		(*Wrap up break Flags to Variable for shipment to UI*)
		ECatSlave_Cable_Breaks.0:= ATV320_NotPresent AND Prev_EcatNode_Present;
		ECatSlave_Cable_Breaks.1:= ATV320_PortB_MissingLink;


(*$$$$$$$$$$$$$$$$$$$$$$$$$$$$$$$$$$$$$$$$$$$$$$$$$$$$Gather All Standard and System Inputs $$$$$$$$$$$$$$$$$$$$$$$$$$$$$$$$$$$$$$$$$$$$$$$$$$$$$$$$$$$$$*)

	(*--------------- System Inputsfrom VFD System Outputs -------------------------*)

	(*Status_Word*)
		Operating_State_Ready:= NOT Status_Word.0;
		Operating_State_Switched_On:=Status_Word.1;
		Operating_State_Operation_enabled:=Status_Word.2;
		Operating_State_Fault:=Status_Word.3;
		Voltage_Enabled:=Status_Word.4;
		Operating_State_Quick_Stop:=Status_Word.5;
		Operating_State_Switch_On_Dissabled:=Status_Word.6;
		Error_Class0:=Status_Word.7;
		Halt_Requested:=Status_Word.8;
		Remote:=Status_Word.9;
		Target_Reached:=Status_Word.10;
		Internal_Limit:=Status_Word.11;
		Operating_Mode_Specific:=Status_Word.12;
		X_ERR:=Status_Word.13;
		X_End:=Status_Word.14;
		Ref_OK:=Status_Word.15;



(*$$$$$$$$$$$$$$$$$$$$$$$$$$$$$$$$$$$$$$$$$$$$$$$$$$ Internal Code $$$$$$$$$$$$$$$$$$$$$$$$$$$$$$$$$$$$$$$$$$$$$$$$$$$$$$$$*)


	(*Capture time between part feeding*)
	Move_TMR(
			IN:= (Enable_Operation AND NOT Operating_State_Switch_On_Dissabled) AND Enable_Motion,
			PT:= T#9999s,
			Q=> ,
			ET=>
			);
	IF Move_TMR.IN
		THEN
			Move_TIME:= Move_TMR.ET;
	END_IF;


(*$$$$$$$$$$$$$$$$$$$$$$$$$$$$$$$$$$$$$$$$$$$$$$ Transfer Standard Outputs $$$$$$$$$$$$$$$$$$$$$$$$$$$$$$$$$$$$$$$$$$$*)

	Discrete_Image.Status_Word:= Status_Word;
	Discrete_Image.Control_Word:= Control_Word;
	Discrete_Image.Target_Velocity:= Target_Velocity;
	Discrete_Image.ECAT_Cable_Breaks:= ECatSlave_Cable_Breaks;

	Discrete_Image.VFD_State:= VFD_State;
	Discrete_Image.Move_TIME:= Move_TIME;



	(*--------------- System Outputs to VFD System Inputs -------------------------*)

	(*Control Word*)
	Control_Word.0:= (Operating_State_Switch_On AND NOT Operating_State_Switch_On_Dissabled) AND Enable_Motion;
	Control_Word.1:= Enable_Voltage AND Enable_Motion;
	Control_Word.2:= Operating_State_Quick_Stop_Req;
	Control_Word.3:= (Enable_Operation AND NOT Operating_State_Switch_On_Dissabled) AND Enable_Motion;
	Control_Word.4:= Operating_Mode_Bit4;
	Control_Word.5:= Operating_Mode_Bit5;
	Control_Word.6:= Operating_Mode_Bit6;
	Control_Word.7:= Fault_Reset;
	Control_Word.8:= Halt;
	Control_Word.9:= Operating_Mode_Bit9;
	Control_Word.10:= FALSE; (*reserved - must be 0*)
	Control_Word.11:= FALSE; (*reserved - must be 0*)
	Control_Word.12:= FALSE; (*reserved - must be 0*)
	Control_Word.13:= FALSE; (*reserved - must be 0*)
	Control_Word.14:= FALSE; (*reserved - must be 0*)
	Control_Word.15:= FALSE; (*reserved - must be 0*)


	(*Output Frequency*)
	IF (Requested_Freq>=0) AND (Requested_Freq<51)
		THEN
			Target_Velocity:= (Requested_Freq * 30);
	ELSE
			Target_Velocity:= 0;
	END_IF;
















(*end*)

END_FUNCTION_BLOCK

// ---- POUs/FBs/FB_GTAC_Ped_20240808.TcPOU
(*!!!!!!!!!!!!!!!!!!!!!!!!!!!!!!!!!!!!!!!!!!!!!!!!!!!!!!!!!!!!!!!!!!!!!!!!!!!!!!!!!!!!!!!!!!!!!!!!!!!!!!!!!!!!!!!!!!!!!!!!!!!!!!!!!!!!!!!!!!!!!!!!!!!!!!!!!!
FB for framework of a generic Ped Station (welding, Sealing, stud welding etc)
	author: Brent Lekx-Toniolo of Sodecia GTAC
	Feb, 2015
--------------------------------------------------------------------------------------------------------------
REVISION NOTES:
	Version: 20150224:
	- Original Concept, b.lekx-toniolo
	Version: 20150426:
	- Change Order of Fix ID, b.lekx-toniolo
	- Added Complete Reset Input
	Version: 20151104:
	- added linkable hardware types, b.lekx-toniolo
	Version: 20160728
	- added control fro brake option, b.lekx-toniolo
	- added configuration inputs for Input node and VB counts, b.lekx-toniolo
	Version: 20160915
	- added "blank_position_checks" Input, b.lekx-toniolo, r.remillard, j.vandongen
	- added "Dresser_Enable" Input, b.lekx-toniolo, r.remillard, j.vandongen
	Version: 20160926
	- Corrected doubled up valve 1 instance, b.lekx-toniolo
	Version 20170404
	- add Part present sensors, j.vandongen
	Version 20170704
	- changed valve instances, j.vandongen
	Version 20170725
	- added VB_Node_Count to UI and updated discrete_image, j.vandongen
	- removed dresser wording form variables to make fb more generic, j.vandongen
	- moved tool_at_positions to outside the fb, j.vandongen
	Version 20170810
	- corrected PP fault issue, j.vandongen
	Version 20220808
	- Added Prev_EcatNode_Present and Prev_EcatNode_ID, c.drees
	Version 20230126
	- Built in SwingArm functionality to combine PEDxx with SwingArmXX, c.drees
	Version 20240514
	- Add in Nodelayout configuration data area, b.lexk-toniolo
	Version 20240808
	- Add in ability to externally control portions of the N50 output block
--------------------------------------------------------------------------------------------------------------
*)

FUNCTION_BLOCK FB_GTAC_Ped_20240808
	VAR_INPUT

		Enable_Prog: BOOL;
		Enable_Motion: BOOL;
		Mode_Select: INT;
		Go_Home: BOOL;
		Reset_Production: BOOL;
		Model_Data: INT;
		Task_Data: UINT;
		Manual_Requests: DINT;
		Dry_Cycle: BOOL;
		Cell_In_Services: BOOL;
		PrevProcess_Complete: BOOL;
		Blank_Position_Checks: BOOL;
		Start_TipDress_Cycle: BOOL;
		Start_TipChange_Cycle: BOOL;
		
		(*Generic Position Variables*)
		Tool_At_Home: BOOL;
		Tool_At_Work0: BOOL;
		Tool_At_Work1: BOOL;

		Part_Present1_REQ: BOOL;
		Part_Present2_REQ: BOOL;
		Part_Present3_REQ: BOOL;
		Part_Present4_REQ: BOOL;

		Work_Robots_Clear: BOOL;
		Work_Robots_WorkingOK: BOOL;
		Work_Robots_Complete: BOOL;
		Work_Robots_LHPartInEOAT: BOOL;
		Work_Robots_RHPartInEOAT: BOOL;
		Work_Robots_CommonPartInEOAT: BOOL;
		Work_Robots_EOATEmpty: BOOL;
	(*Node Counts and configuration data*)
		Input_Node_Count: UDINT;
		Output_Node_Count: UDINT;
			Output_Node_UserREQS: UINT;
		VB_Node_Count: UDINT;
		Part_Present_Count: UDINT;
		Option_SwingCylinder: BOOL;		(*Enables a Cylinder used for changing the Ped Item (Weld gun as example) position OR Tip Dress Swing*)
			Swing_ADV_REQ: BOOL;		
			Swing_RET_REQ: BOOL;
		Option_TipDresser: BOOL;	(*Enables Tip Dresser functionality*)
		Option_TipChanger: BOOL;		(*Enables Tip Changer functionality*)
		NodeLayout:udt_ECATNodeData_20221507;

	(*Ecat configuration*)
	
		Prev_EcatNode_Present:BOOL;
		Prev_EcatNode_ID:STRING;
	END_VAR

	VAR
(*Hardware Related Data Types*)
			(*Develop "Beckhoff Nodes"*)
			{attribute 'OPC.UA.DA':='1'}
			N01 AT %I*: udt_EP1008_002_v2;
			{attribute 'OPC.UA.DA':='1'}
			N02 AT %I*: udt_EP1008_002_v2;
			{attribute 'OPC.UA.DA':='1'}
			N50 AT %Q*: udt_EP2028_002_v2;
			{attribute 'OPC.UA.DA':='1'}
			N50_STAT AT %I*: udt_EP2028_002_STAT;
			{attribute 'OPC.UA.DA':='1'}
			N100 AT %Q*: udt_SMC_EX260_ValveBank;
			{attribute 'OPC.UA.DA':='1'}
			N100_STAT AT %I*:udt_SMC_EX260_Stat;
(* Nodes States*)
		NodeState: ARRAY[0..63] OF UINT;
		DiscreteNode_OK: BOOL;
(*Cable Break States*)
		ECatSlave_Cable_Breaks: ARRAY[0..1] OF DINT;
(*Standard Internal Variables*)

		(*Generic Position Variables*)
		Tool_At_Work: UINT;

		(*General Internals*)
		In_Auto: BOOL;
		In_Manual: BOOL;

		Auto_Run: BOOL;
		Reset_All_Completes:BOOL;

		Start_Work_Robots: BOOL;
		Work_Robots_Proceed: BOOL;

		Prod_Inc: R_TRIG;
		Cycle_Time: TON;
		Cycle_Time_Pulse: R_TRIG;
		CLFaulted: UDINT;
		PPFaulted: UDINT;
		Manual_Ind_HomePrompt: BOOL;

(*Non-Standard Variables*)
		(*FB Instances*)
		Swing1FB: FB_Cylinder_Status;
		Part_Present1FB: FB_PP_Sensor;
		Part_Present2FB: FB_PP_Sensor;
		Part_Present3FB: FB_PP_Sensor;
		Part_Present4FB: FB_PP_Sensor;

		(*Valve FBs*)
		Valve1FB: FB_GTAC_Valve_20170704;
		Valve2FB: FB_GTAC_Valve_20170704;
		(*Tool Positions*)
		Swing1ADVD: BOOL;
		Swing1RETD: BOOL;
		(*Motion Sequence Variables*)
			Clamp_Step: UINT;
			Repo1_Step: UINT;
			Repo2_Step: UINT;
			Repo3_Step: UINT;
			Repo4_Step: UINT;
			Unclamp_Step: UINT;


END_VAR

	(*data that needs to be retained in the event of a power cycle*)
	VAR PERSISTENT
		Working_Complete: BOOL;
		Cycle_Complete: BOOL;
		Production_Count:INT;
		TipDress_Complete: BOOL;
		TipChange_Complete: BOOL;
		Repo_REQS: UINT;
	END_VAR

	VAR_OUTPUT
		Prog_Ok: BOOL;
		Discrete_Image: udt_PEDxx_Image_20240808;
		In_Auto_Mode: BOOL;
		In_Manual_Mode: BOOL;
		Manual_Indicators: DINT;
		At_Home: BOOL;
		CLFaults1:UDINT;
		CLFaults2:UDINT;
		CLFaults3:UDINT;
		CLFaults4:UDINT;
		PPFaults: UDINT;
		Prod_Count_Out: INT;
		Cycle_Time_Out: TIME;
		PrevCycle_Time_Out: TIME;
		Tool_Call_ForWorkRobots: BOOL;
		Robots_Clear_ToProceed: BOOL;
		Task_ID: UINT;
		Fix_ID: UINT;
		Model_ID: UINT;
		Work_Complete_Ack: BOOL;
		Repo_Ack: UINT;

	(*Part Present Sensors*)
		(*Main Body Present*)
		Part_Present1: BOOL;
		Part_Present2: BOOL;
		Part_Present3: BOOL;
		Part_Present4: BOOL;

	END_VAR

	(*Set FB_OK to True*)
	Prog_OK:= TRUE;
(*$$$$$$$$$$$$$$$$$$$$$$$$$$$$$$$$$$$$$$$$$$$$$$$$Gather Status Of Hardware $$$$$$$$$$$$$$$$$$$$$$$$$$$$$$$$$$$$$$$$$$$$$$$$$$$$*)
	(*Discrete I/O Nodes*)
	IF N01.InfoData.State=8 OR (Input_Node_Count<1)
		AND (N02.InfoData.State=8 OR (Input_Node_Count<2))
		AND (N50_STAT.InfoData.State=8 OR (Output_Node_Count<1))
		AND (N100_Stat.InfoData.State=8 OR (VB_Node_Count<1))
			THEN DiscreteNode_OK:=TRUE;
	ELSE DiscreteNode_OK:=FALSE;
	END_IF;
	
	(*Cable Break Detection*)
	ECatSlave_Cable_Breaks[0]:= FUN_GTAC_EcatSlaveConnState
							(N01.InfoData.State,
							N02.InfoData.State,
							N50_STAT.InfoData.State,
							N100_Stat.InfoData.State,
							0,0,0,0,0,0,0,0,0,0,0,0,0,0,0,0,0,0,0,0,0,0,0,0,0,0); (*Function Returns Flags to warn of possible cable break*)

(*$$$$$$$$$$$$$$$$$$$$$$$$$$$$$$$$$$$$$$$$$$$$$ Gather Safety Inputs $$$$$$$$$$$$$$$$$$$$$$$$$$$$$$$$$$$$$$$$$$$$$$$$$$$$$$$$$*)

(*$$$$$$$$$$$$$$$$$$$$$$$$$$$$$$$$$$$$$$$$$$$$$ Gather Standard Inputs $$$$$$$$$$$$$$$$$$$$$$$$$$$$$$$$$$$$$$$$$$$$$$$$$$$$$$$$$*)
	IF Option_SwingCylinder
		THEN
		(*Swing1 - Ped item OR Tip Dresser Swing (if Option_TipDresser is enabled)*)
		Swing1FB(
			Advanced_Sensor:= N01.I.0,
			Retracted_Sensor:= N01.I.1,
			Advance_Solenoid:= N100.Q.0,
			Retract_Solenoid:= N100.Q.1,
			Adv_Delay:= T#0.5S ,
			Ret_Delay:= T#0.5s ,
			Fault_Delay:= T#4s ,
			In_Advanced_Position=> Swing1ADVD,
			In_Retracted_Position=> Swing1RETD,
			Faulted=> CLFaults1.0 );
	ELSIF NOT  Option_SwingCylinder
		THEN
		Swing1ADVD:= FALSE;
		Swing1RETD:= TRUE;
		CLFaults1.0:= FALSE;

	END_IF;

(*$$$$$$$$$$$$$$$$$$$$$$$$$$$$$$$$$$$$$$$$$$$$$$$$ Internal Code $$$$$$$$$$$$$$$$$$$$$$$$$$$$$$$$$$$$$$$$$$$$$$$$$$$$$$$$$$$$$$$$$$$$*)
(*Auto / Manual Mode Code*)
In_Auto:= TRUE;(*FORCED IN AUTO*)

	IF Mode_Select.0 AND NOT Mode_Select.1
		THEN
			In_Auto:= TRUE;
			In_Auto_Mode:= TRUE;
	END_IF;
	IF NOT Mode_Select.0 AND Mode_Select.1
		THEN
			In_Auto:= FALSE;
			In_Auto_Mode:= FALSE;
	END_IF;
	In_Manual:= NOT In_Auto;
	In_Manual_Mode:= In_Manual;

(*--------------------------------------------------------------------------------Tool Positions---------------------------------------------------------------*)
(*+++++++++++THIS AREA IS CUSTOM PER INSTALLATION AND WILL HAVE TO BE MODIFIED PER +++++++++++++*)
(*+++++++++++THIS AREA IS CUSTOM PER INSTALLATION AND WILL HAVE TO BE MODIFIED PER +++++++++++++*)

	Tool_At_Work.0:= Tool_At_Work0;
	Tool_At_Work.1:= Tool_At_Work1;

(*>>>>>>>>>>>>>>>>>>>>>>>>>>>>>>>>>>>>>>>>>> Auto Run Cycle >>>>>>>>>>>>>>>>>>>>>>>>>>>>>>>>>>>>>>>*)
(*+++++++++++THIS AREA IS CUSTOM PER INSTALLATION AND WILL HAVE TO BE MODIFIED PER +++++++++++++*)
(*+++++++++++THIS AREA IS CUSTOM PER INSTALLATION AND WILL HAVE TO BE MODIFIED PER +++++++++++++*)
	(*Control of Auto_Run*)
	Auto_Run:= Enable_Motion AND In_Auto AND Model_Data<>0 AND NOT Cycle_Complete;

	(*Auto Run Enables All Other Auto Cycle Code*)
	IF Auto_Run
		THEN
			IF NOT Working_Complete  AND PrevProcess_Complete
				THEN
					(*Start Work Robots*)
					Start_Work_Robots:= (Work_Robots_CommonPartInEOAT OR Work_Robots_LHPartInEOAT OR Work_Robots_RHPartInEOAT)
										AND (((Tool_At_Work.0 AND NOT Repo_Reqs.0) OR (Tool_At_Work.1 AND Repo_Reqs.0)) OR Blank_Position_Checks)
										AND (Model_Data <> 0);
;					(*Allow Work Robots To Proceed*)
					Work_Robots_Proceed:= (Work_Robots_CommonPartInEOAT OR Work_Robots_LHPartInEOAT OR Work_Robots_RHPartInEOAT)
										AND Tool_At_Work.0 AND NOT Repo_Reqs.0 AND PrevProcess_Complete;
			ELSE
					Start_Work_Robots:= FALSE;
					Work_Robots_Proceed:= FALSE;
			END_IF;

	ELSE
		Start_Work_Robots:= FALSE;
	END_IF;

(*---------------------------------------------------------------Completes----------------------------------------------------*)
	(*Wrok at Ped Complete*)
	IF Work_Robots_Complete
		THEN
		Working_Complete:= TRUE;
	END_IF;

(*!!!!!!!!!!!!!!!!!!!!!!!!!!!!!!!!!!!!!!!!!!!!!!!!!!!!!!!!!!!!!!!!!!!!!!!!!!!!!!!!!!!!!!!!!!!!!!!!! Cycle Complete !!!!!!!!!!!!!!!!!!!!!!!!!!!!!!!!!!!!!!!!!!!!!!!!!!!!!!!!!!!!!!!!!!!!!!!!!!!!!!!!!!!!!!!!!!*)
	(*Set Cycle Complete*)
	IF Auto_Run AND Working_Complete
		THEN Cycle_Complete:= TRUE;
	END_IF;
	(*Reset All Completes*)
	IF Work_Robots_Clear
		THEN
			IF Work_Robots_EOATEmpty
				THEN
					Reset_All_Completes:= TRUE;
			ELSE
					Reset_All_Completes:= FALSE;
			END_IF;
	END_IF;
	(*Perform Actual Reset*)
		IF Reset_All_Completes
			THEN
				Cycle_Complete:= FALSE;
				Working_Complete:= FALSE;
				Reset_All_Completes:= FALSE;
		END_IF;


(*$$$$$$$$$$$$$$$$$$$$$$$$$$$$$$$$$$$ Production Counter $$$$$$$$$$$$$$$$$$$$$$$$$$$$$$$$$$$$$$$$$$*)
	(*Increment Production Counter*)
	Prod_Inc.CLK:= Cycle_Complete;
	Prod_Inc();
	IF Prod_Inc.Q
		THEN
		Production_Count:= Production_Count+1;
	END_IF;
	IF Reset_Production
		THEN
		Production_Count:= 0;
	END_IF;
	Prod_Count_Out:= Production_Count;
(*~~~~~~~~~~~~~~~~~~~~~~~~~~~~~~~~ Cycle Time Counters ~~~~~~~~~~~~~~~~~~~~~~~~~*)
	(*Move Previous To Register*)
	Cycle_Time_Pulse.CLK:= Cycle_Complete;
	Cycle_Time_Pulse();
	IF Cycle_Time_Pulse.Q
		THEN
		PrevCycle_Time_Out:= Cycle_Time_Out;
	END_IF;
	(*Monitor Current Cycle Time*)
		Cycle_Time.PT:= T#9999S;
		Cycle_Time.IN:= NOT Cycle_Time_Pulse.Q ;
		Cycle_Time();
		Cycle_Time_Out:= Cycle_Time.ET;


(*%%%%%%%%%%%%%% Call Robots to Tool and Give Them, Task ID, Fixture ID and Model ID %%%%%%%%%%%%%%%%%*)

	(* Perform Call To Tool*)
	Tool_Call_ForWorkRobots:= Enable_Motion AND (NOT Cell_In_Services OR NOT Work_Robots_Clear)
	 							AND Start_Work_Robots;

	(*Allow Robots to Proceed Into Tool*)
	(*!!!!!This is the final OK to allow Robots Into the Tool Area, So it Better Be Ready!!!!!!!*)
	IF Enable_Motion
		THEN
			IF Work_Robots_Proceed AND Work_Robots_WorkingOK
				THEN Robots_Clear_ToProceed:=TRUE;
			END_IF;
		ELSE Robots_Clear_ToProceed:= FALSE;
	END_IF;

	(*Develop Task IDs - See Global Variable, "TaskID_Record"*)

	IF Start_Work_Robots AND Enable_Motion
		THEN Task_ID:= Task_Data;
	ELSE Task_ID:= 0;
	END_IF;

	(*Develop Fixture ID*)
	IF Work_Robots_CommonPartInEOAT AND NOT Work_Robots_LHPartInEOAT AND NOT Work_Robots_RHPartInEOAT
		THEN
			Fix_ID:= 1;
	ELSIF Work_Robots_LHPartInEOAT AND NOT Work_Robots_RHPartInEOAT AND NOT Work_Robots_CommonPartInEOAT
		THEN
			Fix_ID:= 2;
	ELSIF NOT Work_Robots_LHPartInEOAT AND Work_Robots_RHPartInEOAT AND NOT Work_Robots_CommonPartInEOAT
		THEN
			Fix_ID:= 3;
	ELSE
			Fix_ID:= 0;
	END_IF;
	(*Develop Model ID*)
	Model_ID:=Model_Data;

(*+++++++++++++++++++++++++++++++++++++++++++++++ Task Complete Acks ++++++++++++++++++++++++++*)

	(*Weld Complete Ack*)
	Work_Complete_Ack:= Work_Robots_Complete AND Working_Complete;



(*!!!!!!!!!!!!!!!!!!!!!!!!!!!!!!!!!!!!!!!!!!!!!!!!!!!!!!!!!!!!!!!!!!!!!!!!!!!!!!!!!!!!!!!! Tool Repositions !!!!!!!!!!!!!!!!!!!!!!!!!!!!!!!!!!!!!!!!!!!!!!!!!!!!!!!!!!!!!!!!!!!!!!!!!!!!!!!!!!!!!!!!!!!*)
(*+++++++++++THIS AREA IS CUSTOM PER INSTALLATION AND WILL HAVE TO BE MODIFIED PER +++++++++++++*)
(*+++++++++++THIS AREA IS CUSTOM PER INSTALLATION AND WILL HAVE TO BE MODIFIED PER +++++++++++++*)

	(*Reposition Request#1*)
	IF FALSE
		THEN
			Repo_Reqs.0:= TRUE;
	END_IF;
	(*Reposition Request#2*)
	IF FALSE
		THEN
			Repo_Reqs.1:= TRUE;
	END_IF;
	(*Reposition Request#3*)
	IF FALSE
		THEN
			Repo_Reqs.2:= TRUE;
	END_IF;
	(*Reposition Request#4*)
	IF FALSE
		THEN
			Repo_Reqs.3:= TRUE;
	END_IF;
	(*Reset All Reposition Acks At the End Of Cycle*)
	IF Cycle_Complete
		THEN
			Repo_Reqs:= 0;
	END_IF;
(*------------------------- Reposition Acks ---------------------*)
	Repo_Ack.0:= Repo_Reqs.0 AND FALSE;
	Repo_Ack.1:= Repo_Reqs.0 AND FALSE;
	Repo_Ack.2:= Repo_Reqs.0 AND FALSE;
	Repo_Ack.3:= Repo_Reqs.0 AND FALSE;



(*?????????????????????????????????????????????????????????????????????????????????????????????????????????????????????????????????*)

(*$$$$$$$$$$$$$$$$$$$$$$$$$$$$$$$$$$$$$$$$$$$$$$$$$$$ Faults $$$$$$$$$$$$$$$$$$$$$$$$$$$$$$$$$$$$$$$$$$$$$$$$$$$$$$$*)
	(*Clamp/Cylider Faults Group 1*)
		IF CLFaults1>0
			THEN CLFaulted.1:=TRUE;
		ELSE
			CLFaulted.1:=FALSE;
		END_IF;
	(*Clamp/Cylider Faults Group 2*)
		IF CLFaults2>0
			THEN CLFaulted.2:=TRUE;
		ELSE
			CLFaulted.2:=FALSE;
		END_IF;
	(*Clamp/Cylider Faults Group 3*)
		IF CLFaults3>0
			THEN CLFaulted.3:=TRUE;
		ELSE
			CLFaulted.3:=FALSE;
		END_IF;
	(*Clamp/Cylinder Faults Group 4 - Reserved Flag for QA Check Motion Faults*)
		IF CLFaults4>0
			THEN CLFaulted.4:=TRUE;
		ELSE
			CLFaulted.4:=FALSE;
		END_IF;
	(*Bit 0 is designated as ANY Clamp Group Faulted*)
	IF CLFaulted.1 OR CLFaulted.2 OR CLFaulted.3
		THEN CLFaulted.0:= TRUE;
	ELSE CLFaulted.0 := FALSE;
	END_IF;

	(*Part Present Sensor Faults*)
		IF PPFaults>0
			THEN PPFaulted.0:=TRUE;
		ELSE
			PPFaulted.0:=FALSE;
		END_IF;

(*$$$$$$$$$$$$$$$$$$$$$$$$$$$$$$$$$$$$$$$$$$$$$$ Transfer Standard Outputs $$$$$$$$$$$$$$$$$$$$$$$$$$$$$$$$$$$$$$$$$$$*)

	(*Transfer General Status and I/O Images for Display On UI*)
	Discrete_Image.Input_Node_Count:= Input_Node_Count;
	Discrete_Image.Output_Node_Count:= Output_Node_Count;
	Discrete_Image.VB_Node_Count:= VB_Node_Count;
	Discrete_Image.Option_SwingCylinder:= Option_SwingCylinder;
	Discrete_Image.Option_TipDresser:= Option_TipDresser;
	Discrete_Image.Option_TipChanger:= Option_TipChanger;
	
	Discrete_Image.CLFaults1:= CLFaults1;
	Discrete_Image.CLFaults2:= CLFaults2;
	Discrete_Image.CLFaults3:= CLFaults3;
	Discrete_Image.CLFaults4:= CLFaults4;
	Discrete_Image.CLFaulted:= CLFaulted;
	
	Discrete_Image.PPFaults:= PPFaults;
	Discrete_Image.PPFaulted:= PPFaulted;
	
	
	Discrete_Image.N01:= N01;
	Discrete_Image.N02:= N02;
	Discrete_Image.N50_STAT:= N50_STAT;
	Discrete_Image.N50:= N50;
	Discrete_Image.N100_STAT:= N100_STAT;
	Discrete_Image.N100:= N100;

	Discrete_Image.NodeLayout:= NodeLayout;
	
	
(*-----------------------------------------------------------------------------------------Transfer Discrete Outputs --------------------------------------------------------------------------------*)

	(*N50 Output Block*)
	IF Enable_Motion AND (Output_Node_Count >0) THEN
		IF Option_TipDresser THEN
			N50.Q.0:= FALSE;		(*Dedicated for Dresser Cutter CW*)
			N50.Q.1:= FALSE;		(*Dedicated for Dresser Cutter CCW*)
			N50.Q.2:= Output_Node_UserREQS.2;
			N50.Q.3:= Output_Node_UserREQS.3;
			N50.Q.4:= Output_Node_UserREQS.4;
			N50.Q.5:= Output_Node_UserREQS.5;
			N50.Q.6:= Output_Node_UserREQS.6;
			N50.Q.7:= Output_Node_UserREQS.7;
		ELSE
			N50.Q.0:= Output_Node_UserREQS.0;
			N50.Q.1:= Output_Node_UserREQS.1;
			N50.Q.2:= Output_Node_UserREQS.2;
			N50.Q.3:= Output_Node_UserREQS.3;
			N50.Q.4:= Output_Node_UserREQS.4;
			N50.Q.5:= Output_Node_UserREQS.5;
			N50.Q.6:= Output_Node_UserREQS.6;
			N50.Q.7:= Output_Node_UserREQS.7;
		END_IF;
	ELSE
		N50.Q:= 0;	
	END_IF;
	
	
(*-----------------------------------------------------------------------------------------Transfer Valve Outputs --------------------------------------------------------------------------------*)

	(*Valve 1, A+B*)
	(*Swing Cylinder 1*)
		Valve1FB
			(
			Enable_Motion:= Enable_Motion AND Option_SwingCylinder,
			Enable_Latch:= TRUE,					(*Enabling Runs Valve as detent type (maintained solenoids*)
			Enable_SideA_PreCharge:= FALSE,		(*Enabling Turns Side A PreCharge Active, reset when Side B is energized in Auto*)
			Enable_SideB_PreCharge:= FALSE,		(*Enabling Turns Side B PreCharge Active, reset when Side A is energized in Auto*)
			PreCharge_Time:= T#0.1S,
			Enable_Auto_Commands:= In_Auto,
			In_Auto_SideA_Command:= Swing_ADV_REQ,
			In_Auto_SideB_Command:= Swing_RET_REQ ,
			Enable_Manual_Commands:= In_Manual,
			In_Manual_SideA_Command:= FALSE,
			In_Manual_SideB_Command:= FALSE,
			SideA_Indicator:= Tool_At_Work.0,
			SideB_Indicator:= Tool_At_Work.1,
			TurnOn_SideA_SOL=> N100.Q.0,
			TurnOn_SideB_SOL=> N100.Q.1,
			TurnOn_SideA_Indicator=> Manual_Indicators.0,
			TurnOn_SideB_Indicator=> Manual_Indicators.1
			 );


(*$$$$$$$$$$$$$$$$$$$$$$$$$$$$$$$$$$$$$$$$$$$$$$ Transfer Safety Outputs $$$$$$$$$$$$$$$$$$$$$$$$$$$$$$$$$$$$$$$$$$$*)

END_FUNCTION_BLOCK

// ---- POUs/FBs/FB_Cylinder_Status.TcPOU
(*FB for replacement of typical clamp fault checking code":
	Original Author(s): Brent Lekx-Toniolo of Toniolo Research & Development Inc.; 
	August 2010; version 3.0


------------------------------------------------------------------------------------------
REVISION NOTES:
	Version 20170615
		-  Added disable fault input, b.lekx-toniolo / j.bysma

------------------------------------------------------------------------------------------
*)
FUNCTION_BLOCK FB_Cylinder_Status

	VAR_INPUT
		Enable_FB: BOOL;
		Advanced_Sensor: BOOL;
		Retracted_Sensor: BOOL;
		Advance_Solenoid: BOOL;
		Retract_Solenoid: BOOL;
		Adv_Delay: TIME;
		Ret_Delay: TIME;
		Fault_Delay: TIME;
		Disable_Fault: BOOL;
	END_VAR

	VAR
		At_Advanced: BOOL;
		At_Retracted: BOOL;
		Adv_Delay_TMR: TON;
		Ret_Delay_TMR: TON;
		Sensor_FLT_TMR: TON;
		Advancing_FLT_TMR: TON;
		Retracting_FLT_TMR: TON;
	END_VAR

	VAR_OUTPUT
		FB_OK: BOOL;
		In_Advanced_Position: BOOL;
		In_Retracted_Position: BOOL;
		Faulted: BOOL;
		Sensor_Fault: BOOL;
		Advancing_Fault: BOOL;
		Retracting_Fault: BOOL;
	END_VAR

	(*Set FB_OK to True*)
	FB_OK:= TRUE;
(*$$$$$$$$$$$$$$$$$$$$$$$$$$$$$$$$$$ Internal Code $$$$$$$$$$$$$$$$$$$$$$$$$$$$$$$$$$$$$$$$$$$$$$$*)
	(*Develop Advanced Position*)
	At_Advanced:=Advanced_Sensor AND NOT Retracted_Sensor;

	(*Develop Retracted Position*)
	At_Retracted:=Retracted_Sensor AND NOT Advanced_Sensor;

	(*Delay Advanced Position Output*)
	Adv_Delay_TMR.PT:=Adv_Delay;
	Adv_Delay_TMR.IN:=At_Advanced;
	Adv_Delay_TMR();
	In_Advanced_Position:=Adv_Delay_TMR.Q;

	(*Delay Retracted Position Output*)
	Ret_Delay_TMR.PT:=Ret_Delay;
	Ret_Delay_TMR.IN:=At_Retracted;
	Ret_Delay_TMR();
	In_Retracted_Position:=Ret_Delay_TMR.Q;

(*$$$$$$$$$$$$$$$$$$$$$$$$$$$$$$$$$$$$$$$$ Fault Code $$$$$$$$$$$$$$$$$$$$$$$$$$$$$$$$$$$$$$$$$$$$$$$$*)
	(*Sensor Fault*)
	Sensor_FLT_TMR.PT:=Fault_Delay;
	Sensor_FLT_TMR.IN:=(NOT At_Advanced AND NOT At_Retracted) OR (At_Advanced AND At_Retracted);
	Sensor_FLT_TMR();
	Sensor_Fault:=Sensor_FLT_TMR.Q;

	(*Advancing Fault*)
	Advancing_FLT_TMR.PT:=Fault_Delay;
	Advancing_FLT_TMR.IN:=Advance_Solenoid AND NOT At_Advanced AND NOT Sensor_Fault;
	Advancing_FLT_TMR();
	Advancing_Fault:=Advancing_FLT_TMR.Q;

	(*Retracting Fault*)
	Retracting_FLT_TMR.PT:=Fault_Delay;
	Retracting_FLT_TMR.IN:=Retract_Solenoid AND NOT At_Retracted AND NOT Sensor_Fault;
	Retracting_FLT_TMR();
	Retracting_Fault:=Retracting_FLT_TMR.Q;

	(*Develop Fault Output*)
	Faulted:= NOT Disable_Fault AND (Sensor_Fault OR Advancing_Fault OR Retracting_Fault);

END_FUNCTION_BLOCK

// ---- POUs/FBs/FB_PP_Sensor.TcPOU
(*FB for replacement of typical part present sesnors fault checking
	Original Author(s):. Brent Lekx-Toniolo of Toniolo Research & Development Inc.; 
	August 2010; version 2.0*)


FUNCTION_BLOCK FB_PP_Sensor
VAR_INPUT
		Enable_FB: BOOL;
		Sensor_Input: BOOL;
		On_Trigger1: BOOL;
		On_Trigger2: BOOL;
		Off_Trigger1: BOOL;
		Off_Trigger2: BOOL;
		Disable_Faults: BOOL;
		Fault_Delay: TIME;
END_VAR
VAR
		NotON_FLT_TMR: TON;
		NotOFF_FLT_TMR: TON;

END_VAR

VAR_OUTPUT
		FB_OK: BOOL;
		Status: BOOL;
		Faulted: BOOL;
		NotON_Fault: BOOL;
		NotOFF_Fault: BOOL;
END_VAR

	(*Set FB_OK to True*)
	FB_OK:= TRUE;
(*$$$$$$$$$$$$$$$$$$$$$$$$$$$$$$$$$$ Internal Code $$$$$$$$$$$$$$$$$$$$$$$$$$$$$$$$$$$$$$$$$$$$$$$*)
	(*Pass Status Straight Thru*)
	Status:= Sensor_Input;

	(*Pass Faults*)
	Faulted:= NotON_Fault OR NotOff_Fault;

	(*Develop Not On When Required Fault*)
	NotOn_FLT_TMR.PT:= Fault_Delay;
	NotOn_FLT_TMR.IN:= On_Trigger1 AND On_Trigger2 AND NOT Sensor_Input AND NOT Disable_Faults;
	NotOn_FLT_TMR();
	NotOn_Fault:= NotOn_FLT_TMR.Q;

	(*Develop Not Off When Required Fault*)
	NotOff_FLT_TMR.PT:= Fault_Delay;
	NotOff_FLT_TMR.IN:= Off_Trigger1 AND Off_Trigger2 AND Sensor_Input AND NOT Disable_Faults;
	NotOff_FLT_TMR();
	NotOff_Fault:= NotOff_FLT_TMR.Q;

END_FUNCTION_BLOCK

// ---- POUs/FBs/FB_GTAC_Valve_20170704.TcPOU
(*FB for use with standard double sided Solenoid Valve:
	Original Author(s): Brent Lekx-Toniolo of Sodecia GTAC; 
------------------------------------------------------------------------------------------
REVISION NOTES:
	Version 20150218
	- Original Concept, b.lekx-toniolo (S.H.H.D.I.)
	Version 20160407
	- Added Enable Latch (Detent Type) functionality, r.remillard
	Version 20170704
	-incorporated precharge into the function block, j.vandongen

------------------------------------------------------------------------------------------
*)


FUNCTION_BLOCK FB_GTAC_Valve_20170704

VAR_INPUT
	Enable_Motion: BOOL;
	Enable_Auto_Commands: BOOL;
	Enable_Latch: BOOL;									(*Used to maintain Solenoid at last requested state*)
	Enable_SideA_PreCharge: BOOL;
	Enable_SideB_PreCharge: BOOL;
	In_Auto_SideA_Command: BOOL;
	In_Auto_SideB_Command: BOOL;
	Enable_Manual_Commands: BOOL;
	In_Manual_SideA_Command: BOOL;
	In_Manual_SideB_Command: BOOL;
	SideA_Indicator: BOOL;
	SideB_Indicator: BOOL;
	PreCharge_Time: TIME;
END_VAR

VAR
	In_Auto_SideA_REQ: BOOL;
	In_Auto_SideB_REQ: BOOL;
	In_Manual_SideA_REQ: BOOL;
	In_Manual_SideB_REQ: BOOL;
	PreCharge_Timer_SideA: TON;
	PreCharge_Timer_SideB: TON;
END_VAR

VAR_OUTPUT
	TurnOn_SideA_SOL: BOOL;
	TurnOn_SideB_SOL: BOOL;
	TurnOn_SideA_Indicator: BOOL;
	TurnOn_SideB_Indicator: BOOL;

END_VAR

(*Gather Auto Mode Requests*)
	In_Auto_SideA_REQ:= Enable_Motion AND Enable_Auto_Commands AND In_Auto_SideA_Command;
	In_Auto_SideB_REQ:= Enable_Motion AND Enable_Auto_Commands AND In_Auto_SideB_Command;



(*Gather Manual Mode Requests*)
	In_Manual_SideA_REQ:= Enable_Motion AND Enable_Manual_Commands AND In_Manual_SideA_Command;
	In_Manual_SideB_REQ:= Enable_Motion AND Enable_Manual_Commands AND In_Manual_SideB_Command;



(*Pre Charge Timers*)
	PreCharge_Timer_SideA(
					In:= Enable_SideA_PreCharge AND (In_Auto_SideA_REQ OR (PreCharge_Timer_SideA.Q AND NOT In_Auto_SideB_REQ)),
					PT:= PreCharge_Time
					);

	PreCharge_Timer_SideB(
					In:= Enable_SideB_PreCharge AND (In_Auto_SideB_REQ OR (PreCharge_Timer_SideA.Q AND NOT In_Auto_SideA_REQ)),
					PT:= PreCharge_Time
					);



(*Set Actual Outputs*)
	(*Valve Outputs*)
	TurnOn_SideA_SOL:= (((In_Auto_SideA_REQ AND (PreCharge_Timer_SideA.Q OR NOT Enable_SideA_PreCharge))
						OR (In_Auto_SideB_REQ AND NOT PreCharge_Timer_SideB.Q AND Enable_SideB_PreCharge)
						OR In_Manual_SideA_REQ)
						OR (Enable_Latch AND TurnOn_SideA_SOL AND NOT (In_Auto_SideB_REQ OR In_Manual_SideB_REQ)))
						AND NOT TurnOn_SideB_SOL;

	TurnOn_SideB_SOL:= (((In_Auto_SideB_REQ AND (PreCharge_Timer_SideB.Q OR NOT Enable_SideB_PreCharge))
						OR (In_Auto_SideA_REQ AND NOT PreCharge_Timer_SideA.Q AND Enable_SideA_PreCharge)
						 OR In_Manual_SideB_REQ)
						OR (Enable_Latch AND TurnOn_SideB_SOL AND NOT (In_Auto_SideA_REQ OR In_Manual_SideA_REQ)))
						AND NOT TurnOn_SideA_SOL;



	(*Indicator Outputs*)
	TurnOn_SideA_Indicator:= SideA_Indicator;
	TurnOn_SideB_Indicator:= SideB_Indicator;



















(*end*)

END_FUNCTION_BLOCK

// ---- POUs/FBs/FB_VertiGuard_20260310.TcPOU

FUNCTION_BLOCK FB_VertiGuard_20260310

VAR_INPUT
	
		Enable_FB: BOOL;
		Enable_Motion: BOOL;
		Enable_Latch: BOOL;

		GateClose_REQ: BOOL;		(*Request to close the door*)
		GateOpen_REQ: BOOL;			(*Request to open the door*)
		
		GateOpened_Time: TIME;		(*Door Open Fault Control Timer*)
		GateClosed_Time: TIME;		(*Door Closed Fault Control Timer*)
		
		GateOpen_Precharge_Time: TIME;	(*Pre Charge Time For Opening Gate*)

		GateClosed_Switches: BOOL;	(*Switches to detect Door Closed*)
		GateOpened_Switches: BOOL;	(*Switches to detect Door opened*)

		Fault_Time: TIME;
		
END_VAR

VAR
	
		Gate_CloseSR: SR; 					(*Latch to Close the door*)
		Gate_OpenSR: SR;					(*Latch to Open the door*)

		GateOpen_Precharge_TMR: TON; 		(*Pre Charge Timer For Opening The Gate*)
		GateOpened_TMR: TON;				(*Timer to say gate is open, no door open switches*)
		GateClosed_TMR: TON;				(*Timer to say gate is closed*)

		Fault_TMR: TON;

END_VAR

VAR_OUTPUT

		FB_OK: BOOL;

		GateClose_CMD: BOOL;	(*Command the door to close*)
		GateOpen_CMD: BOOL;		(*Command the door to open*)
		Gate_Closed: BOOL;		(*Door is closed*)
		Gate_Opened: BOOL;		(*Door is open*)

		Faulted: BOOL;	

END_VAR

(*Set FB_OK to True*)
	FB_OK:= TRUE;

	(*Set Gate to Close*)
	Gate_CloseSR(
			SET1:= Enable_Latch AND GateClose_REQ AND NOT GateOpen_REQ,
			RESET:= NOT Enable_Latch OR (GateOpen_REQ AND Gate_Closed),
			Q1=>
			);

	(*Set Gate to Open*)
	Gate_OpenSR(
			SET1:= Enable_Motion AND Enable_Latch AND GateOpen_REQ AND NOT GateClose_REQ,
			RESET:= NOT Enable_Motion OR NOT Enable_Latch OR (GateClose_REQ OR Gate_Opened),
			Q1=>
			);

	(*Pre Charge Timer For Opening Guard*)
	GateOpen_Precharge_TMR(
					In:= Enable_Motion AND ((Enable_Latch AND Gate_OpenSR.Q1) OR (NOT Enable_Latch AND GateOpen_REQ)),
					PT:= GateOpen_Precharge_Time
					);

	(*Set Actual Outputs*)
	(*Valve Outputs*)
	(*Note ------> The closed state has a pin lock so at the moment the gate is closed, we cancel the latch*)
	GateClose_CMD:= (((Enable_Latch AND Gate_CloseSR.Q1 (*AND NOT Gate_Closed*)) OR (NOT Enable_Latch AND GateClose_REQ)) AND NOT ((Enable_Latch AND Gate_OpenSR.Q1) OR (NOT Enable_Latch AND GateOpen_REQ)))
					OR (((Enable_Latch AND Gate_OpenSR.Q1) OR (NOT Enable_Latch AND GateOpen_REQ)) AND NOT GateOpen_Precharge_TMR.Q);
	GateOpen_CMD:= Enable_Motion AND GateOpen_Precharge_TMR.Q AND ((Enable_Latch AND Gate_OpenSR.Q1) OR (NOT Enable_Latch AND GateOpen_REQ)) AND NOT ((Enable_Latch AND Gate_CloseSR.Q1) OR (NOT Enable_Latch AND GateClose_REQ));
					
	(*Gate Opened Timer*)
	GateOpened_TMR(
			IN:= GateOpened_Switches AND GateOpen_CMD,
			PT:= GateOpened_Time,
			Q=> ,
			ET=>
			);

	(*Gate Closed Timer*)
	GateClosed_TMR(
			IN:= GateClosed_Switches,
			PT:= GateClosed_Time,
			Q=> ,
			ET=>
			);

	(*Capture Gate Status*)
	IF GateClosed_Switches AND GateClosed_TMR.Q
		THEN
			Gate_Closed:= TRUE;
			Gate_Opened:= FALSE;
	ELSIF GateOpened_Switches AND GateOpened_TMR.Q
		THEN
			Gate_Closed:= FALSE;
			Gate_Opened:= TRUE;
	END_IF;
	
	(*Capture Gate Faults*)
	Fault_TMR(
			IN:= (GateClose_CMD AND NOT Gate_Closed) OR (GateOpen_CMD AND NOT Gate_Opened),
			PT:= Fault_Time,
			Q=> Faulted,
			ET=> );


(*end*)

END_FUNCTION_BLOCK

// ---- POUs/GTAC_CONFIG.TcPOU
(* FOR USE BY SODECIA GTAC ONLY !!!*)
(* Sodecia GTAC Configuration data for this particular machine*)

(*----------------------------------------------------------------------------------------------------------------------
REVISION NOTES: 
	Date: Dec 2019
	- Added PROD_CONFIG action and modified production code for R&D request, b.lekx-toniolo/r.remillard
	Date: Jan 2021
	- Automated Machine Serial Variable, b.lekx-toniolo
	Date: Oct 2021
	- Updated serial section for new engineering serial format changes, b.lekx-toniolo
	Date: Feb 2024
	- Added In_Sim_Mode for simulation integration, b.lekx-toniolo
	Date: Sept 2024
	- Added MD component, b.lekx-toniolo
	Date: November 2024
	- PD to IS rename, as per GH SSCC610 repo Issue#162, b.lekx-toniolo

------------------------------------------------------------------------------------------------------------------------*)



PROGRAM GTAC_CONFIG
VAR
		(*Machine Specific Information: Serial Number, Comon Name, Build Level Used, Application Devloper*)
		Machine_Serial: STRING;
		Machine_Common_Name: STRING;
		Machine_Build_Used: STRING;
		Machine_Appl_Dev: STRING;
		
		(*Production Reporting Configuration Data*)
		ProdConfig_Target_CycleTime: TIME;
		ProdConfig_Common: udt_Generic_ShiftCommonConfig_20220420;
		ProdConfig_Day: udt_Generic_ShiftConfigTOD_20160527;
		ProdConfig_Aft: udt_Generic_ShiftConfigTOD_20160527;
		ProdConfig_Mid: udt_Generic_ShiftConfigTOD_20160527;

		ProdConfig_OK: BOOL;
		ProdConfig_Source_FLT: BOOL;
		ProdConfig_Option_SelectInShiftChange: BOOL;

		(*Config Data (For Use to Configure Code Directives)*)
		Option_EL6900_TemperatureHighLimit: INT;

		Option_Air1: BOOL;
		Option_Air2: BOOL;

		Option_Water1: BOOL;
		Option_Water2: BOOL;

		Option_WaterTimeOut_Enable: BOOL;
		Option_WaterFlowTimeOut_SP: TIME;
		Option_WaterTempHighLimit1: REAL;
		Option_WaterFlowLowLimit1: REAL;
		Option_WaterTempHighLimit2: REAL;
		Option_WaterFlowLowLimit2: REAL;

		Option_ESW_Count: UINT;

		Option_IS_Count: UINT;
		Option_IC_Count: UINT;
		Option_HumanFix_Enables: UDINT;
		Option_InternalFix_Count: UINT;
		Option_Robot_Count: UINT;
		Option_Ped_Count: UINT;
		Option_StudController_Count: UINT;
		Option_SealController_Count: UINT;
		Option_NutWelder_Count: UINT;
		(*Option_EOAT_Count: UINT;*)
		Option_LaserController_Count: UINT;
		Option_SD_Count: UINT;
		Option_MD_Count: UINT;
		Option_VFD_Count: UINT;
		Option_EP9214_Count: UINT;
		(*General Development State Modes for Cell*)
		Dry_Cycle_Enabled: BOOL;			(*Place Machine Into Dry Cycle (Ignore PP Sensors)*)
		Local_DryCycle_Enables: UDINT;	(*Used to place individual fixtures into Dry Cycle*)
		Low_Speed_Enabled: BOOL;		(*Set All Robots and Drives to Low Speed Mode*)
		Under_Construction: BOOL; 			(*Set Machine Into Construction Mode for Easier Teaching Etc !!!! Use with Caution !!!!*)
		In_SIM_Mode: BOOL;					(*Set machine into Sim mode during simulation development*)


		(*Configuration Fault Flag*)
		Fault: UDINT;


	Report_Trigger_ACKS: INT;
END_VAR

(*$$$$$$$$$$$$ Set Data As required to configure the machine $$$$$$$$$$$$$$$$$$$$*)

(*-----------------------------------------Machine / Application Specific Information-----------------------------------*)

(*NOTE: Machine Serial is now automatically read from the project name, simply rename your project elements for your machine and we'll do the rest!*)
	Machine_Serial:= FUN_GTAC_ReturnSetLengthSTR(Out_To_ICxx.Appdata.ProjectName, 22);

(*NOTE: Change to a common use name that the customer will recognize*)
	Machine_Common_Name:= 'Volvo Truck V2004 Front Bumper';
	
(*NOTE: When you started with a server copy of the FW the software came in a folder called All_yyymmdd_state*) 
	(*use this for below and change the value below only once upon creating this application, this takes a snap shot of the FW build level you started with*)
	Machine_Build_Used:= 'All_20250506_release';
	
(*NOTE: Be sure to Enter your name or initials here, if mulitple application developers worked on the project then list all*)
	Machine_Appl_Dev:= 'w.griffiths, r.jone, b.lekx-toniolo';
		

(*---------------------------------------Production Report Configuration -----------------------------------*)
(*Machine Target Cycle Time (can also be set individually at each fixture, see Fixture -> Production Action*)
(*Changes per Model ID - All controlled by Fixture 01*)

(*504*)
	IF (Fix01.Model_ID=1) THEN
		ProdConfig_Target_CycleTime:=T#156S;
(*524*)
	ELSIF (Fix01.Model_ID=2) THEN
		ProdConfig_Target_CycleTime:=T#184.8S;
(*543*)
	ELSIF (Fix01.Model_ID=3) THEN
		ProdConfig_Target_CycleTime:=T#136.1S;
(*526 OR 536*)
	ELSIF (Fix01.Model_ID=4) OR (Fix01.Model_ID=5) THEN
		ProdConfig_Target_CycleTime:=T#221S;
(*550 OR 571*)
	ELSIF (Fix01.Model_ID=6) OR (Fix01.Model_ID=7) THEN
		ProdConfig_Target_CycleTime:= T#251S;
	END_IF
	
	

(*Call Prod_Config_Constraints Action*)
	PROD_CONFIG_Constraints();

(*Call Prod_Config Action*)
	PROD_CONFIG();
	
(*Call Reports Action*)
	REPORTS();	

(*Call SIM Action*)
	SIM();	

(*-----------------------------------------Machine Configuration Options -----------------------------------*)
(*Select to Check for 1st MAIN Air Manifold Faults*)
	Option_Air1:= TRUE;
(*Select to Check for 2nd MAIN Air Manifold Faults*)
	Option_Air2:= FALSE;

(*Select to Check for 1st MAIN Water Manifold Faults*)
	Option_Water1:= FALSE;
(*Select to Check for 2nd MAIN Water Manifold Faults*)
	Option_Water2:= FALSE;

(*Global Water Setpoints*)
	Option_WaterTimeOut_Enable:= NOT Under_Construction AND
									TRUE;		(*Enable Robot Water Flow Timeout Feature (Stop Water flow if flow not achived after setpoint)*)
	Option_WaterFlowTimeOut_SP:= T#5.5S;			(*Setpoint for Robot Water Flow Timeout feature, 1.0s Min, 10.0s Max*)
	Option_WaterTempHighLimit1:= 24;
	Option_WaterTempHighLimit2:= 24;

	Option_WaterFlowLowLimit1:= 5;
	Option_WaterFlowLowLimit2:= 5;


(*Select Amount of Enable Switches will be present in Machine 0 Min, 4 max*)
	Option_ESW_Count:= 3;

(*Select Amount of IS cabinets for machine 1 min, CURRENTLY, DO NOT EXCEED 1*)
	Option_IS_Count:= 1;
(*Select Amount of ICs for machine 1 min, 8 max*)
	Option_IC_Count:= 3;
(*Set Enable Bits for  Human Fixtures for machine*)
	Option_HumanFix_Enables.1:= TRUE; 		(*Enable Human Fix01 on IC01*)
	Option_HumanFix_Enables.2:= TRUE; 		(*Enable Human Fix02 on IC01*)
	Option_HumanFix_Enables.3:= TRUE; 		(*Enable Human Fix03 on IC02*)
	Option_HumanFix_Enables.4:= TRUE; 		(*Enable Human Fix04 on IC02*)
	Option_HumanFix_Enables.5:= TRUE; 		(*Enable Human Fix05 on IC03*)
	Option_HumanFix_Enables.6:= FALSE; 		(*Enable Human Fix06 on IC03*)
	Option_HumanFix_Enables.7:= FALSE; 		(*Enable Human Fix07 on IC04*)
	Option_HumanFix_Enables.8:= FALSE; 		(*Enable Human Fix08 on IC04*)
	Option_HumanFix_Enables.9:= FALSE; 		(*Enable Human Fix09 on IC05*)
	Option_HumanFix_Enables.10:= FALSE; 		(*Enable Human Fix10 on IC05*)
	Option_HumanFix_Enables.11:= FALSE; 		(*Enable Human Fix11 on IC06*)
	Option_HumanFix_Enables.12:= FALSE; 		(*Enable Human Fix12 on IC06*)
	Option_HumanFix_Enables.13:= FALSE; 		(*Enable Human Fix13 on IC07*)
	Option_HumanFix_Enables.14:= FALSE; 		(*Enable Human Fix14 on IC07*)
	Option_HumanFix_Enables.15:= FALSE; 		(*Enable Human Fix15 on IC08*)
	Option_HumanFix_Enables.16:= FALSE; 		(*Enable Human Fix16 on IC08*)

(*Select Amount of Internal Fixtures for machine 0 min, 12 max (check config)*)
	Option_InternalFix_Count:= 5;

(*Select Amount of Robots for machine 1 min, 30 max*)
	Option_Robot_Count:= 11;

(*Select Amount of EOAT for machine 0 min, 10 max*)
	(*Set EOAT Amount under each robot*)

(*Select Amount of Spot Weld Peds for machine 0 min, 30 max*)
	Option_Ped_Count:= 0;	//Maybe 1 for marking but aiming for Fixture

(*Select Amount of Stud Weld Controllers for machine 0 min, 10 max*)
	Option_StudController_Count:= 0;

(*Select Amount of Sealant Controllers for machine 0 min, 10 max*)
	Option_SealController_Count:= 0;

(*Select Amount of Nut Welder Systems for machine 0 min, 5 max*)
	Option_NutWelder_Count:= 0;

(*Select Amount of Laser Control Systems for machine 0 min, 9 max*)
	Option_LaserController_Count:= 0;

(*Select Amount of Servo Drives (SD) for machine 0 min, 30 max*)
	Option_SD_Count:= 0;
(*Select Amount of Motorized Doors will be present in Machine 0 Min, 5 max*)
	Option_MD_Count:= 2;
(*Select Amount of VFDs that will be present in Machine 0 Min, 5 max*)
	Option_VFD_Count:= 2;
(*Select Amount of 9214 that will be present in Machine 0 Min, 3 max*)
	Option_EP9214_Count:= 0;

(*-----------------------------------------Machine Development Operational States-----------------------------------*)

(*Dry Cycle*)
	Dry_Cycle_Enabled:= In_From_ICxx.Enable_Dry_Cycle;				(*Global Dry Cycle Enable*)
	Local_DryCycle_Enables:= In_From_ICxx.Local_DryCycle_Enables; 	(*Fixture by Fixture Dry Cycle Enables*)

(*Low Speed Mode*)
	Low_Speed_Enabled:= In_From_ICxx.Low_Speed_Req;

(*!!!!!!!!!!!Under Construction Bit for Temp Use Only During Integration!!!!!!!!!!!!!!*)
(*!!!!!!!!!!!Under Construction Bit for Temp Use Only During Integration!!!!!!!!!!!!!!*)
(*!!!!!!!!!!!Under Construction Bit for Temp Use Only During Integration!!!!!!!!!!!!!!*)
(* Blanks Robot Water Faults, Bypasses all Robot to Robot Software teach Interlocks and Allows Operation with no Robot TQM or Collision Detect*)

	Under_Construction:= FALSE; (*DEBUG, set to false after finished construction of machine*)

(*!!!!!!!!!!!Under Construction Bit for Temp Use Only During Integration!!!!!!!!!!!!!!*)
(*!!!!!!!!!!!Under Construction Bit for Temp Use Only During Integration!!!!!!!!!!!!!!*)
(*!!!!!!!!!!!Under Construction Bit for Temp Use Only During Integration!!!!!!!!!!!!!!*)



(*!!!!!!!!!!!In Simulation Mode for Temp Use Only During Simulation!!!!!!!!!!!!!!*)
(*!!!!!!!!!!!In Simulation Mode for Temp Use Only During Simulation!!!!!!!!!!!!!!*)
(*!!!!!!!!!!!In Simulation Mode for Temp Use Only During Simulation!!!!!!!!!!!!!*)
(* Reroutes a number of I/O points to be exchanged with Simulation environment (via OPC) instead of physical I/O*) 

	In_SIM_Mode:= FALSE; (*DEBUG, set to false after simulation work is done and you're onto a physical machine*)

(*!!!!!!!!!!!In Simulation Mode for Temp Use Only During Simulation!!!!!!!!!!!!!!*)
(*!!!!!!!!!!!In Simulation Mode for Temp Use Only During Simulation!!!!!!!!!!!!!!*)
(*!!!!!!!!!!!In Simulation Mode for Temp Use Only During Simulation!!!!!!!!!!!!!!*)


(*---------------------------------------------- Check Configuration Data ------------------------------------------------------*)

	(*Check Shift Time Configuration Basics*)

	Fault.1:= NOT ProdConfig_OK;

	Fault.2:= Option_WaterFlowTimeOut_SP<T#1.0s OR Option_WaterFlowTimeOut_SP>T#10.0s;
	Fault.3:= Option_WaterTempHighLimit1>30 OR Option_WaterTempHighLimit2>30
			OR Option_WaterFlowLowLimit1<3 OR Option_WaterFlowLowLimit2<3;
	Fault.4:= (Option_IS_Count <1 OR Option_IS_Count >1);
	Fault.5:= (Option_ESW_Count <0 OR Option_ESW_Count >4);
	Fault.6:= (Option_IC_Count <1 OR Option_IC_Count >8);
	Fault.7:= (Option_HumanFix_Enables <2 OR Option_HumanFix_Enables >131070);
	Fault.8:= ((Option_HumanFix_Enables.3 OR Option_HumanFix_Enables.4)  AND (Option_IC_Count <2)) OR
			((Option_HumanFix_Enables.5 OR Option_HumanFix_Enables.6)  AND (Option_IC_Count <3)) OR
			((Option_HumanFix_Enables.7 OR Option_HumanFix_Enables.8)  AND (Option_IC_Count <4)) OR
			((Option_HumanFix_Enables.9 OR Option_HumanFix_Enables.10)  AND (Option_IC_Count <5)) OR
			((Option_HumanFix_Enables.11 OR Option_HumanFix_Enables.12)  AND (Option_IC_Count <6)) OR
			((Option_HumanFix_Enables.13 OR Option_HumanFix_Enables.14)  AND (Option_IC_Count <7)) OR
			((Option_HumanFix_Enables.15 OR Option_HumanFix_Enables.16)  AND (Option_IC_Count <8));
	Fault.9:= (Option_InternalFix_Count <0 OR Option_InternalFix_Count >9);
	Fault.10:= (Option_Robot_Count <1 OR Option_Robot_Count >30);
	Fault.11:= (Option_Ped_Count <0 OR Option_Ped_Count >30);
	Fault.12:= (Option_StudController_Count <0 OR Option_StudController_Count >10);
	Fault.13:= (Option_SealController_Count <0 OR Option_SealController_Count >10);
	Fault.14:= (Option_NutWelder_Count <0 OR Option_NutWelder_Count >5);
	Fault.15:= FALSE;	(*Used to be EOAT*)
	Fault.16:= (Option_LaserController_Count <0 OR Option_LaserController_Count >9);
	Fault.17:= (Option_SD_Count<0 OR Option_SD_Count>30);
	Fault.18:= (Option_MD_Count<0 OR Option_MD_Count>5);
	Fault.30:= MAIN.ECAT_Master.Config_SlaveCount_ExceedsMax_FLT; 								(*Check Sys_Man Confgured Slave Count vs Maximum amount permissable in FB_GTAC_EtherCATMaster_yyyymmdd (see brent)*)
	(*Set General Configuration Faulted Flag*)
	Fault.0:= Fault.1OR Fault.2 OR Fault.3 OR Fault.4
			OR Fault.5 OR Fault.6 OR Fault.7 OR Fault.8
			OR Fault.9 OR Fault.10 OR Fault.11 OR Fault.12
			OR Fault.13 OR Fault.14 OR Fault.15 OR Fault.16
			OR Fault.17 OR Fault.18
			OR Fault.30;

ACTION PROD_CONFIG:
(*------------------------------------------------------------------------------------------------------------------------*)
(* ------------------------------------------- Production Configuration --------------------------------------*)
(*------------------------------------------------------------------------------------------------------------------------*)

(*Change Configuration data source depending on user selection on UI*)

(*0 = set production config source as default (GTAC default Config)*)
IF In_From_ICxx_Pers.ProdConfig_Common.Config_Source = 0
	OR In_From_ICxx_Pers.ProdConfig_Common.ResetProdConfig_To_Default
	THEN
		ProdConfig_Source_FLT:= FALSE;
		ProdConfig_Common.Shift_Enables:=14; (*bit.0 = not used, bit.1 = Day Enabled, bit.2 = Aft Enabled, bit.3 = Mid Enabled*)
		ProdConfig_Common.Break_Count:= 3;
		ProdConfig_Common.Config_Option_Flags.0:= TRUE;	(*Force In_Shift_Change option flag, leave other option flags*)
		(*Machine Shift and Breaks Setup*)
			(*Day Shift*)
			ProdConfig_Day.Shift_StartTime:= TOD#7:00:00;
				ProdConfig_Day.Break1_StartTime:= TOD#9:00:00;
				ProdConfig_Day.Break1_EndTime:= TOD#9:10:00;
				ProdConfig_Day.Break2_StartTime:= TOD#12:00:00;
				ProdConfig_Day.Break2_EndTime:= TOD#12:30:00;
				ProdConfig_Day.Break3_StartTime:= TOD#13:30:00;
				ProdConfig_Day.Break3_EndTime:= TOD#13:40:00;
			ProdConfig_Day.Shift_EndTime:= TOD#15:00:00;



			(*Afternoon Shift*)
			ProdConfig_Aft.Shift_StartTime:= TOD#15:00:00;
				ProdConfig_Aft.Break1_StartTime:= TOD#17:00:00;
				ProdConfig_Aft.Break1_EndTime:= TOD#17:10:00;
				ProdConfig_Aft.Break2_StartTime:= TOD#20:00:00;
				ProdConfig_Aft.Break2_EndTime:= TOD#20:30:00;
				ProdConfig_Aft.Break3_StartTime:= TOD#21:30:00;
				ProdConfig_Aft.Break3_EndTime:= TOD#21:40:00;
			ProdConfig_Aft.Shift_EndTime:= TOD#23:00:00;

			(*Midnight Shift*)
			ProdConfig_Mid.Shift_StartTime:= TOD#23:00:00;
				ProdConfig_Mid.Break1_StartTime:= TOD#1:00:00;
				ProdConfig_Mid.Break1_EndTime:= TOD#1:10:00;
				ProdConfig_Mid.Break2_StartTime:= TOD#4:00:00;
				ProdConfig_Mid.Break2_EndTime:= TOD#4:30:00;
				ProdConfig_Mid.Break3_StartTime:= TOD#5:30:00;
				ProdConfig_Mid.Break3_EndTime:= TOD#5:40:00;
			ProdConfig_Mid.Shift_EndTime:= TOD#7:00:00;

 (*1 = set production config source as via UI (User Set Config)*)
ELSIF In_From_ICxx_Pers.ProdConfig_Common.Config_Source = 1 AND
		NOT In_From_ICxx_Pers.ProdConfig_Common.ResetProdConfig_To_Default
	THEN
		ProdConfig_Source_FLT:= FALSE;
		ProdConfig_Common.Shift_Enables:= In_From_ICxx_Pers.ProdConfig_Common.Shift_Enables;
		ProdConfig_Common.Break_Count:= In_From_ICxx_Pers.ProdConfig_Common.Break_Count;
		ProdConfig_Common.Config_Option_Flags:= In_From_ICxx_Pers.ProdConfig_Common.Config_Option_Flags;
		(*Machine Shift and Breaks Setup*)
			(*Day Shift*)
			ProdConfig_Day.Shift_StartTime:= UDINT_TO_TOD(In_From_ICxx_Pers.ProdConfig_Day.Shift_StartTime);
				ProdConfig_Day.Break1_StartTime:= UDINT_TO_TOD(In_From_ICxx_Pers.ProdConfig_Day.Break1_StartTime);
				ProdConfig_Day.Break1_EndTime:= UDINT_TO_TOD(In_From_ICxx_Pers.ProdConfig_Day.Break1_EndTime);
				ProdConfig_Day.Break2_StartTime:= UDINT_TO_TOD(In_From_ICxx_Pers.ProdConfig_Day.Break2_StartTime);
				ProdConfig_Day.Break2_EndTime:= UDINT_TO_TOD(In_From_ICxx_Pers.ProdConfig_Day.Break2_EndTime);
				ProdConfig_Day.Break3_StartTime:= UDINT_TO_TOD(In_From_ICxx_Pers.ProdConfig_Day.Break3_StartTime);
				ProdConfig_Day.Break3_EndTime:= UDINT_TO_TOD(In_From_ICxx_Pers.ProdConfig_Day.Break3_EndTime);
			ProdConfig_Day.Shift_EndTime:= UDINT_TO_TOD(In_From_ICxx_Pers.ProdConfig_Day.Shift_EndTime);

			(*Afternoon Shift*)
			ProdConfig_Aft.Shift_StartTime:= UDINT_TO_TOD(In_From_ICxx_Pers.ProdConfig_Aft.Shift_StartTime);
				ProdConfig_Aft.Break1_StartTime:= UDINT_TO_TOD(In_From_ICxx_Pers.ProdConfig_Aft.Break1_StartTime);
				ProdConfig_Aft.Break1_EndTime:= UDINT_TO_TOD(In_From_ICxx_Pers.ProdConfig_Aft.Break1_EndTime);
				ProdConfig_Aft.Break2_StartTime:= UDINT_TO_TOD(In_From_ICxx_Pers.ProdConfig_Aft.Break2_StartTime);
				ProdConfig_Aft.Break2_EndTime:= UDINT_TO_TOD(In_From_ICxx_Pers.ProdConfig_Aft.Break2_EndTime);
				ProdConfig_Aft.Break3_StartTime:= UDINT_TO_TOD(In_From_ICxx_Pers.ProdConfig_Aft.Break3_StartTime);
				ProdConfig_Aft.Break3_EndTime:= UDINT_TO_TOD(In_From_ICxx_Pers.ProdConfig_Aft.Break3_EndTime);
			ProdConfig_Aft.Shift_EndTime:= UDINT_TO_TOD(In_From_ICxx_Pers.ProdConfig_Aft.Shift_EndTime);

			(*Midnight Shift*)
			ProdConfig_Mid.Shift_StartTime:= UDINT_TO_TOD(In_From_ICxx_Pers.ProdConfig_Mid.Shift_StartTime);
				ProdConfig_Mid.Break1_StartTime:= UDINT_TO_TOD(In_From_ICxx_Pers.ProdConfig_Mid.Break1_StartTime);
				ProdConfig_Mid.Break1_EndTime:= UDINT_TO_TOD(In_From_ICxx_Pers.ProdConfig_Mid.Break1_EndTime);
				ProdConfig_Mid.Break2_StartTime:= UDINT_TO_TOD(In_From_ICxx_Pers.ProdConfig_Mid.Break2_StartTime);
				ProdConfig_Mid.Break2_EndTime:= UDINT_TO_TOD(In_From_ICxx_Pers.ProdConfig_Mid.Break2_EndTime);
				ProdConfig_Mid.Break3_StartTime:= UDINT_TO_TOD(In_From_ICxx_Pers.ProdConfig_Mid.Break3_StartTime);
				ProdConfig_Mid.Break3_EndTime:= UDINT_TO_TOD(In_From_ICxx_Pers.ProdConfig_Mid.Break3_EndTime);
			ProdConfig_Mid.Shift_EndTime:= UDINT_TO_TOD(In_From_ICxx_Pers.ProdConfig_Mid.Shift_EndTime);
ELSE
	ProdConfig_Source_FLT:= TRUE;

END_IF;

(*--------------------------------------------------------------- Check that config data is ok ---------------------------------------------------*)
	ProdConfig_OK:= NOT ProdConfig_Source_FLT AND
					(Fix01.Production_Report.FB_Ok OR NOT Option_HumanFix_Enables.1) AND
					(Fix02.Production_Report.FB_Ok OR NOT Option_HumanFix_Enables.2) AND
					(Fix03.Production_Report.FB_Ok OR NOT Option_HumanFix_Enables.3) AND
					(Fix04.Production_Report.FB_Ok OR NOT Option_HumanFix_Enables.4) AND
					(Fix05.Production_Report.FB_Ok OR NOT Option_HumanFix_Enables.5) AND
					(Fix06.Production_Report.FB_Ok OR NOT Option_HumanFix_Enables.6) AND
					(Fix07.Production_Report.FB_Ok OR NOT Option_HumanFix_Enables.7) AND
					(Fix07.Production_Report.FB_Ok OR NOT Option_HumanFix_Enables.8) AND
					(Fix09.Production_Report.FB_Ok OR NOT Option_HumanFix_Enables.9) AND
					(Fix10.Production_Report.FB_Ok OR NOT Option_HumanFix_Enables.10) AND
					(Fix11.Production_Report.FB_Ok OR NOT Option_HumanFix_Enables.11) AND
					(Fix12.Production_Report.FB_Ok OR NOT Option_HumanFix_Enables.12) AND
					(Fix13.Production_Report.FB_Ok OR NOT Option_HumanFix_Enables.13) AND
					(Fix14.Production_Report.FB_Ok OR NOT Option_HumanFix_Enables.14) AND
					(Fix15.Production_Report.FB_Ok OR NOT Option_HumanFix_Enables.15) AND
					(Fix16.Production_Report.FB_Ok OR NOT Option_HumanFix_Enables.16) AND
					(Fix101.Production_Report.FB_Ok OR (Option_InternalFix_Count<1)) AND
					(Fix102.Production_Report.FB_Ok OR (Option_InternalFix_Count<2)) AND
					(Fix103.Production_Report.FB_Ok OR (Option_InternalFix_Count<3)) AND
					(Fix104.Production_Report.FB_Ok OR (Option_InternalFix_Count<4)) AND
					(Fix105.Production_Report.FB_Ok OR (Option_InternalFix_Count<5)) AND
					(Fix106.Production_Report.FB_Ok OR (Option_InternalFix_Count<6)) AND
					(Fix107.Production_Report.FB_Ok OR (Option_InternalFix_Count<7)) AND
					(Fix108.Production_Report.FB_Ok OR (Option_InternalFix_Count<8)) AND
					(Fix109.Production_Report.FB_Ok OR (Option_InternalFix_Count<9)) AND
					(Fix110.Production_Report.FB_Ok OR (Option_InternalFix_Count<10)) AND
					(Fix111.Production_Report.FB_Ok OR (Option_InternalFix_Count<11)) AND
					(Fix112.Production_Report.FB_Ok OR (Option_InternalFix_Count<12));

(*------------------------------------------------------------------- Map Outputs of Config -------------------------------------------------------*)
	ProdConfig_Option_SelectInShiftChange:= ProdConfig_Common.Config_Option_Flags.0;

(*-----------------------------------------------------------------------------------------------------------------------------------------------------*)
(*Load User Config with GTAC Default data if this is the first boot and no user data has been configured or if user selects to reset to defaults*)



IF	(MAIN.Starting_Scan_Pulse AND
	In_From_ICxx_Pers.ProdConfig_Common.Config_Source = 0 AND 					(*0 = set production config source as default (GTAC default Config)*)
	In_From_ICxx_Pers.ProdConfig_Day.Shift_StartTime=0 AND
	In_From_ICxx_Pers.ProdConfig_Aft.Shift_StartTime=0 AND
	In_From_ICxx_Pers.ProdConfig_Mid.Shift_StartTime=0)
	OR
	(In_From_ICxx_Pers.ProdConfig_Common.Config_Source = 1 AND				(*1 = set production config source as via UI (User Set Config)*)
	In_From_ICxx_Pers.ProdConfig_Common.ResetProdConfig_To_Default)
	THEN
		(*Set config data common to all shifts*)
		In_From_ICxx_Pers.ProdConfig_Common.Shift_Enables:= ProdConfig_Common.Shift_Enables;
		In_From_ICxx_Pers.ProdConfig_Common.Break_Count:= ProdConfig_Common.Break_Count;
		In_From_ICxx_Pers.ProdConfig_Common.Config_Option_Flags.0:= TRUE; (*Set In_Shift_Change option flag, leave other option flags*)
		In_From_ICxx_Pers.ProdConfig_Common.Config_Option_Flags.10:= FALSE; (*Reset File save type option flag, leave other option flags*)

		(*Set shift specfic config data*)
			(*Day Shift*)
			In_From_ICxx_Pers.ProdConfig_Day.Shift_StartTime:= TOD_TO_UDINT(ProdConfig_Day.Shift_StartTime);
				In_From_ICxx_Pers.ProdConfig_Day.Break1_StartTime:= TOD_TO_UDINT(ProdConfig_Day.Break1_StartTime);
				In_From_ICxx_Pers.ProdConfig_Day.Break1_EndTime:= TOD_TO_UDINT(ProdConfig_Day.Break1_EndTime);
				In_From_ICxx_Pers.ProdConfig_Day.Break2_StartTime:= TOD_TO_UDINT(ProdConfig_Day.Break2_StartTime);
				In_From_ICxx_Pers.ProdConfig_Day.Break2_EndTime:= TOD_TO_UDINT(ProdConfig_Day.Break2_EndTime);
				In_From_ICxx_Pers.ProdConfig_Day.Break3_StartTime:= TOD_TO_UDINT(ProdConfig_Day.Break3_StartTime);
				In_From_ICxx_Pers.ProdConfig_Day.Break3_EndTime:= TOD_TO_UDINT(ProdConfig_Day.Break3_EndTime);
			In_From_ICxx_Pers.ProdConfig_Day.Shift_EndTime:= TOD_TO_UDINT(ProdConfig_Day.Shift_EndTime);
			(*Aft Shift*)
			In_From_ICxx_Pers.ProdConfig_Aft.Shift_StartTime:= TOD_TO_UDINT(ProdConfig_Aft.Shift_StartTime);
				In_From_ICxx_Pers.ProdConfig_Aft.Break1_StartTime:= TOD_TO_UDINT(ProdConfig_Aft.Break1_StartTime);
				In_From_ICxx_Pers.ProdConfig_Aft.Break1_EndTime:= TOD_TO_UDINT(ProdConfig_Aft.Break1_EndTime);
				In_From_ICxx_Pers.ProdConfig_Aft.Break2_StartTime:= TOD_TO_UDINT(ProdConfig_Aft.Break2_StartTime);
				In_From_ICxx_Pers.ProdConfig_Aft.Break2_EndTime:= TOD_TO_UDINT(ProdConfig_Aft.Break2_EndTime);
				In_From_ICxx_Pers.ProdConfig_Aft.Break3_StartTime:= TOD_TO_UDINT(ProdConfig_Aft.Break3_StartTime);
				In_From_ICxx_Pers.ProdConfig_Aft.Break3_EndTime:= TOD_TO_UDINT(ProdConfig_Aft.Break3_EndTime);
			In_From_ICxx_Pers.ProdConfig_Aft.Shift_EndTime:= TOD_TO_UDINT(ProdConfig_Aft.Shift_EndTime);
			(*Mid Shift*)
			In_From_ICxx_Pers.ProdConfig_Mid.Shift_StartTime:= TOD_TO_UDINT(ProdConfig_Mid.Shift_StartTime);
				In_From_ICxx_Pers.ProdConfig_Mid.Break1_StartTime:= TOD_TO_UDINT(ProdConfig_Mid.Break1_StartTime);
				In_From_ICxx_Pers.ProdConfig_Mid.Break1_EndTime:= TOD_TO_UDINT(ProdConfig_Mid.Break1_EndTime);
				In_From_ICxx_Pers.ProdConfig_Mid.Break2_StartTime:= TOD_TO_UDINT(ProdConfig_Mid.Break2_StartTime);
				In_From_ICxx_Pers.ProdConfig_Mid.Break2_EndTime:= TOD_TO_UDINT(ProdConfig_Mid.Break2_EndTime);
				In_From_ICxx_Pers.ProdConfig_Mid.Break3_StartTime:= TOD_TO_UDINT(ProdConfig_Mid.Break3_StartTime);
				In_From_ICxx_Pers.ProdConfig_Mid.Break3_EndTime:= TOD_TO_UDINT(ProdConfig_Mid.Break3_EndTime);
			In_From_ICxx_Pers.ProdConfig_Mid.Shift_EndTime:= TOD_TO_UDINT(ProdConfig_Mid.Shift_EndTime);

END_IF;
END_ACTION

ACTION PROD_CONFIG_Constraints:
(*--------------------------------------------------------------------------------------------------------------------------------------------------------*)
(* ------------------------- Production Configuration Hard Coded Constraints-----------------------------------------------------*)
(*-- Can be changed if require, by user familiar with inner workings of FB_Production_Report_yyyymmdd --*)
(*---------------------------------------------------------------------------------------------------------------------------------------------------------*)


(*----------- Dat Shift Set Constaints -----------*)
	(*Day Shift start must fall between 3am -11am*)
	IF UDINT_TO_TOD(In_From_ICxx_Pers.ProdConfig_Day.Shift_StartTime) < TOD#3:00:00
		THEN
				In_From_ICxx_Pers.ProdConfig_Day.Shift_StartTime:= TOD_TO_UDINT(TOD#3:00:00);

	ELSIF UDINT_TO_TOD(In_From_ICxx_Pers.ProdConfig_Day.Shift_StartTime) > TOD#11:00:00
		THEN
				In_From_ICxx_Pers.ProdConfig_Day.Shift_StartTime:= TOD_TO_UDINT(TOD#11:00:00);

	(*Set Shift minimum span as 1 hour*)
	(*Expand towards next shift*)
	ELSIF (In_From_ICxx_Pers.ProdConfig_Day.Shift_EndTime < (In_From_ICxx_Pers.ProdConfig_Day.Shift_StartTime + 3600000))
			AND (In_From_ICxx_Pers.ProdConfig_Day.Shift_EndTime < In_From_ICxx_Pers.ProdConfig_Aft.Shift_StartTime -3600000)
		THEN
				In_From_ICxx_Pers.ProdConfig_Day.Shift_EndTime:= In_From_ICxx_Pers.ProdConfig_Day.Shift_StartTime + 3600000;
	(*Expand towards previous shift*)
	ELSIF (In_From_ICxx_Pers.ProdConfig_Day.Shift_EndTime < (In_From_ICxx_Pers.ProdConfig_Day.Shift_StartTime + 3600000))
			AND (In_From_ICxx_Pers.ProdConfig_Day.Shift_StartTime > In_From_ICxx_Pers.ProdConfig_Mid.Shift_EndTime +3600000)
		THEN
				In_From_ICxx_Pers.ProdConfig_Day.Shift_StartTime:= In_From_ICxx_Pers.ProdConfig_Day.Shift_EndTime - 3600000;

	(*Set Shift maximum span as 12 hours*)
	ELSIF In_From_ICxx_Pers.ProdConfig_Day.Shift_EndTime > (In_From_ICxx_Pers.ProdConfig_Day.Shift_StartTime + 43200000)
		THEN
				In_From_ICxx_Pers.ProdConfig_Day.Shift_EndTime:= (In_From_ICxx_Pers.ProdConfig_Day.Shift_StartTime + 43200000);

	END_IF;

	(*Break 1 Constraints*)
		(*Start of Break*)
		IF In_From_ICxx_Pers.ProdConfig_Day.Break1_StartTime < In_From_ICxx_Pers.ProdConfig_Day.Shift_StartTime + TOD_TO_UDINT(TOD#00:05:00)
			THEN
				In_From_ICxx_Pers.ProdConfig_Day.Break1_StartTime:= In_From_ICxx_Pers.ProdConfig_Day.Shift_StartTime + TOD_TO_UDINT(TOD#00:05:00);
		ELSIF In_From_ICxx_Pers.ProdConfig_Day.Break1_StartTime > In_From_ICxx_Pers.ProdConfig_Day.Shift_EndTime - TOD_TO_UDINT(TOD#00:30:00)
			THEN
				In_From_ICxx_Pers.ProdConfig_Day.Break1_StartTime:= In_From_ICxx_Pers.ProdConfig_Day.Shift_EndTime - TOD_TO_UDINT(TOD#00:30:00);
		(*Allow Break start time to be pushed by break end time*)
		ELSIF In_From_ICxx_Pers.ProdConfig_Day.Break1_StartTime > In_From_ICxx_Pers.ProdConfig_Day.Break1_EndTime
			THEN
				In_From_ICxx_Pers.ProdConfig_Day.Break1_StartTime:= In_From_ICxx_Pers.ProdConfig_Day.Break1_EndTime - TOD_TO_UDINT(TOD#00:05:00);
		END_IF;

		(*End of Break*)
		IF In_From_ICxx_Pers.ProdConfig_Day.Break1_EndTime < In_From_ICxx_Pers.ProdConfig_Day.Shift_StartTime + TOD_TO_UDINT(TOD#00:10:00)
			THEN
				In_From_ICxx_Pers.ProdConfig_Day.Break1_EndTime:= In_From_ICxx_Pers.ProdConfig_Day.Shift_StartTime + TOD_TO_UDINT(TOD#00:10:00);
		ELSIF In_From_ICxx_Pers.ProdConfig_Day.Break1_EndTime > In_From_ICxx_Pers.ProdConfig_Day.Shift_EndTime - TOD_TO_UDINT(TOD#00:25:00)
			THEN
				In_From_ICxx_Pers.ProdConfig_Day.Break1_EndTime:= In_From_ICxx_Pers.ProdConfig_Day.Shift_EndTime - TOD_TO_UDINT(TOD#00:25:00);
		(*Allow Break end time to be pushed by break start time*)
		ELSIF In_From_ICxx_Pers.ProdConfig_Day.Break1_EndTime < In_From_ICxx_Pers.ProdConfig_Day.Break1_StartTime + TOD_TO_UDINT(TOD#00:05:00)
			THEN
				In_From_ICxx_Pers.ProdConfig_Day.Break1_EndTime:= In_From_ICxx_Pers.ProdConfig_Day.Break1_StartTime + TOD_TO_UDINT(TOD#00:05:00);
		ELSIF In_From_ICxx_Pers.ProdConfig_Day.Break1_EndTime > In_From_ICxx_Pers.ProdConfig_Day.Break2_StartTime - TOD_TO_UDINT(TOD#00:05:00)
			THEN
				In_From_ICxx_Pers.ProdConfig_Day.Break1_EndTime:= In_From_ICxx_Pers.ProdConfig_Day.Break2_StartTime - TOD_TO_UDINT(TOD#00:05:00);
		END_IF;

	(*Break 2 Constraints*)
		(*Start of Break*)
		IF In_From_ICxx_Pers.ProdConfig_Day.Break2_StartTime < In_From_ICxx_Pers.ProdConfig_Day.Shift_StartTime + TOD_TO_UDINT(TOD#00:15:00)
			THEN
				In_From_ICxx_Pers.ProdConfig_Day.Break2_StartTime:= In_From_ICxx_Pers.ProdConfig_Day.Shift_StartTime + TOD_TO_UDINT(TOD#00:15:00);
		ELSIF In_From_ICxx_Pers.ProdConfig_Day.Break2_StartTime > In_From_ICxx_Pers.ProdConfig_Day.Shift_EndTime - TOD_TO_UDINT(TOD#00:20:00)
			THEN
				In_From_ICxx_Pers.ProdConfig_Day.Break2_StartTime:= In_From_ICxx_Pers.ProdConfig_Day.Shift_EndTime - TOD_TO_UDINT(TOD#00:20:00);
		ELSIF In_From_ICxx_Pers.ProdConfig_Day.Break2_StartTime < In_From_ICxx_Pers.ProdConfig_Day.Break1_EndTime + TOD_TO_UDINT(TOD#00:05:00)
			THEN
				In_From_ICxx_Pers.ProdConfig_Day.Break2_StartTime:= In_From_ICxx_Pers.ProdConfig_Day.Break1_EndTime + TOD_TO_UDINT(TOD#00:05:00);
		(*Allow Break start time to be pushed by break end time*)
		ELSIF In_From_ICxx_Pers.ProdConfig_Day.Break2_StartTime > In_From_ICxx_Pers.ProdConfig_Day.Break2_EndTime
			THEN
				In_From_ICxx_Pers.ProdConfig_Day.Break2_StartTime:= In_From_ICxx_Pers.ProdConfig_Day.Break2_EndTime - TOD_TO_UDINT(TOD#00:05:00);
		END_IF;

		(*End of Break*)
		IF In_From_ICxx_Pers.ProdConfig_Day.Break2_EndTime < In_From_ICxx_Pers.ProdConfig_Day.Shift_StartTime + TOD_TO_UDINT(TOD#00:20:00)
			THEN
				In_From_ICxx_Pers.ProdConfig_Day.Break2_EndTime:= In_From_ICxx_Pers.ProdConfig_Day.Shift_StartTime + TOD_TO_UDINT(TOD#00:20:00);
		ELSIF In_From_ICxx_Pers.ProdConfig_Day.Break2_EndTime > In_From_ICxx_Pers.ProdConfig_Day.Shift_EndTime - TOD_TO_UDINT(TOD#00:15:00)
			THEN
				In_From_ICxx_Pers.ProdConfig_Day.Break2_EndTime:= In_From_ICxx_Pers.ProdConfig_Day.Shift_EndTime - TOD_TO_UDINT(TOD#00:15:00);
		(*Allow Break end time to be pushed by break start time*)
		ELSIF In_From_ICxx_Pers.ProdConfig_Day.Break2_EndTime < In_From_ICxx_Pers.ProdConfig_Day.Break2_StartTime + TOD_TO_UDINT(TOD#00:05:00)
			THEN
				In_From_ICxx_Pers.ProdConfig_Day.Break2_EndTime:= In_From_ICxx_Pers.ProdConfig_Day.Break2_StartTime + TOD_TO_UDINT(TOD#00:05:00);
		ELSIF In_From_ICxx_Pers.ProdConfig_Day.Break2_EndTime > In_From_ICxx_Pers.ProdConfig_Day.Break3_StartTime - TOD_TO_UDINT(TOD#00:05:00)
			THEN
				In_From_ICxx_Pers.ProdConfig_Day.Break2_EndTime:= In_From_ICxx_Pers.ProdConfig_Day.Break3_StartTime - TOD_TO_UDINT(TOD#00:05:00);
		END_IF;

	(*Break 3 Constraints*)
		(*Start of Break*)
		IF In_From_ICxx_Pers.ProdConfig_Day.Break3_StartTime < In_From_ICxx_Pers.ProdConfig_Day.Shift_StartTime + TOD_TO_UDINT(TOD#00:20:00)
			THEN
				In_From_ICxx_Pers.ProdConfig_Day.Break3_StartTime:= In_From_ICxx_Pers.ProdConfig_Day.Shift_StartTime + TOD_TO_UDINT(TOD#00:20:00);
		ELSIF In_From_ICxx_Pers.ProdConfig_Day.Break3_StartTime > In_From_ICxx_Pers.ProdConfig_Day.Shift_EndTime - TOD_TO_UDINT(TOD#00:10:00)
			THEN
				In_From_ICxx_Pers.ProdConfig_Day.Break3_StartTime:= In_From_ICxx_Pers.ProdConfig_Day.Shift_EndTime - TOD_TO_UDINT(TOD#00:10:00);
		ELSIF In_From_ICxx_Pers.ProdConfig_Day.Break3_StartTime < In_From_ICxx_Pers.ProdConfig_Day.Break2_EndTime + TOD_TO_UDINT(TOD#00:05:00)
			THEN
				In_From_ICxx_Pers.ProdConfig_Day.Break3_StartTime:= In_From_ICxx_Pers.ProdConfig_Day.Break2_EndTime + TOD_TO_UDINT(TOD#00:05:00);
		(*Allow Break start time to be pushed by break end time*)
		ELSIF In_From_ICxx_Pers.ProdConfig_Day.Break3_StartTime > In_From_ICxx_Pers.ProdConfig_Day.Break3_EndTime
			THEN
				In_From_ICxx_Pers.ProdConfig_Day.Break3_StartTime:= In_From_ICxx_Pers.ProdConfig_Day.Break3_EndTime - TOD_TO_UDINT(TOD#00:05:00);
		END_IF;

		(*End of Break*)
		IF In_From_ICxx_Pers.ProdConfig_Day.Break3_EndTime < In_From_ICxx_Pers.ProdConfig_Day.Shift_StartTime + TOD_TO_UDINT(TOD#00:25:00)
			THEN
				In_From_ICxx_Pers.ProdConfig_Day.Break3_EndTime:= In_From_ICxx_Pers.ProdConfig_Day.Shift_StartTime + TOD_TO_UDINT(TOD#00:25:00);
		ELSIF In_From_ICxx_Pers.ProdConfig_Day.Break3_EndTime > In_From_ICxx_Pers.ProdConfig_Day.Shift_EndTime - TOD_TO_UDINT(TOD#00:05:00)
			THEN
				In_From_ICxx_Pers.ProdConfig_Day.Break3_EndTime:= In_From_ICxx_Pers.ProdConfig_Day.Shift_EndTime - TOD_TO_UDINT(TOD#00:05:00);
		(*Allow Break end time to be pushed by break start time*)
		ELSIF In_From_ICxx_Pers.ProdConfig_Day.Break3_EndTime < In_From_ICxx_Pers.ProdConfig_Day.Break3_StartTime + TOD_TO_UDINT(TOD#00:05:00)
			THEN
				In_From_ICxx_Pers.ProdConfig_Day.Break3_EndTime:= In_From_ICxx_Pers.ProdConfig_Day.Break3_StartTime + TOD_TO_UDINT(TOD#00:05:00);
		END_IF;


(*---------- Set Afternoon Shift Constaints -------------*)
	(*Aft Shift start must fall between 11am -7pm*)
	IF UDINT_TO_TOD(In_From_ICxx_Pers.ProdConfig_Aft.Shift_StartTime) < TOD#11:00:00
		THEN
				In_From_ICxx_Pers.ProdConfig_Aft.Shift_StartTime:= TOD_TO_UDINT(TOD#11:00:00);

	ELSIF UDINT_TO_TOD(In_From_ICxx_Pers.ProdConfig_Aft.Shift_StartTime) > TOD#19:00:00
		THEN
				In_From_ICxx_Pers.ProdConfig_Aft.Shift_StartTime:= TOD_TO_UDINT(TOD#19:00:00);

	(*Set Shift minimum span as 1 hour*)
	(*Expand towards next shift*)
	ELSIF (In_From_ICxx_Pers.ProdConfig_Aft.Shift_EndTime < (In_From_ICxx_Pers.ProdConfig_Aft.Shift_StartTime + 3600000))
			AND (In_From_ICxx_Pers.ProdConfig_Aft.Shift_EndTime < In_From_ICxx_Pers.ProdConfig_Mid.Shift_StartTime -3600000)
		THEN
				In_From_ICxx_Pers.ProdConfig_Aft.Shift_EndTime:= In_From_ICxx_Pers.ProdConfig_Aft.Shift_StartTime + 3600000;
	(*Expand towards previous shift*)
	ELSIF (In_From_ICxx_Pers.ProdConfig_Aft.Shift_EndTime < (In_From_ICxx_Pers.ProdConfig_Aft.Shift_StartTime + 3600000))
			AND (In_From_ICxx_Pers.ProdConfig_Aft.Shift_StartTime > In_From_ICxx_Pers.ProdConfig_Day.Shift_EndTime +3600000)
		THEN
				In_From_ICxx_Pers.ProdConfig_Aft.Shift_StartTime:= In_From_ICxx_Pers.ProdConfig_Aft.Shift_EndTime - 3600000;
		(*Extra push scenario to avoid Aft shift getting boxed in by Days and Mids scenario*)
		ELSIF (In_From_ICxx_Pers.ProdConfig_Aft.Shift_EndTime < (In_From_ICxx_Pers.ProdConfig_Aft.Shift_StartTime + 3600000))
				AND (In_From_ICxx_Pers.ProdConfig_Aft.Shift_EndTime > In_From_ICxx_Pers.ProdConfig_Mid.Shift_StartTime -3600000)
				AND In_From_ICxx_Pers.ProdConfig_Mid.Shift_StartTime < (TOD_TO_UDINT(TOD#23:00:00) -3600000)
			THEN
					In_From_ICxx_Pers.ProdConfig_Mid.Shift_StartTime:= In_From_ICxx_Pers.ProdConfig_Aft.Shift_StartTime + 3600000;
					In_From_ICxx_Pers.ProdConfig_Aft.Shift_EndTime:= In_From_ICxx_Pers.ProdConfig_Aft.Shift_StartTime + 3600000;
	(*Set Shift maximum span as 12 hours*)
	ELSIF In_From_ICxx_Pers.ProdConfig_Aft.Shift_EndTime  >= (In_From_ICxx_Pers.ProdConfig_Aft.Shift_StartTime + 43200000)
		THEN
				In_From_ICxx_Pers.ProdConfig_Aft.Shift_EndTime:= (In_From_ICxx_Pers.ProdConfig_Aft.Shift_StartTime + 43200000);

	(*Set Aft Shift maximum end time as 23:59:00 (only midnight shift shall roll over midnight)*)
	ELSIF UDINT_TO_TOD(In_From_ICxx_Pers.ProdConfig_Aft.Shift_EndTime)  > TOD#23:59:00
		THEN
				In_From_ICxx_Pers.ProdConfig_Aft.Shift_EndTime:= TOD_TO_UDINT(TOD#23:59:00);

	END_IF;

	(*Break 1 Constraints*)
		(*Start of Break*)
		IF In_From_ICxx_Pers.ProdConfig_Aft.Break1_StartTime < In_From_ICxx_Pers.ProdConfig_Aft.Shift_StartTime + TOD_TO_UDINT(TOD#00:05:00)
			THEN
				In_From_ICxx_Pers.ProdConfig_Aft.Break1_StartTime:= In_From_ICxx_Pers.ProdConfig_Aft.Shift_StartTime + TOD_TO_UDINT(TOD#00:05:00);
		ELSIF In_From_ICxx_Pers.ProdConfig_Aft.Break1_StartTime > In_From_ICxx_Pers.ProdConfig_Aft.Shift_EndTime - TOD_TO_UDINT(TOD#00:30:00)
			THEN
				In_From_ICxx_Pers.ProdConfig_Aft.Break1_StartTime:= In_From_ICxx_Pers.ProdConfig_Aft.Shift_EndTime - TOD_TO_UDINT(TOD#00:30:00);
		(*Allow Break start time to be pushed by break end time*)
		ELSIF In_From_ICxx_Pers.ProdConfig_Aft.Break1_StartTime > In_From_ICxx_Pers.ProdConfig_Aft.Break1_EndTime
			THEN
				In_From_ICxx_Pers.ProdConfig_Aft.Break1_StartTime:= In_From_ICxx_Pers.ProdConfig_Aft.Break1_EndTime - TOD_TO_UDINT(TOD#00:05:00);
		END_IF;

		(*End of Break*)
		IF In_From_ICxx_Pers.ProdConfig_Aft.Break1_EndTime < In_From_ICxx_Pers.ProdConfig_Aft.Shift_StartTime + TOD_TO_UDINT(TOD#00:10:00)
			THEN
				In_From_ICxx_Pers.ProdConfig_Aft.Break1_EndTime:= In_From_ICxx_Pers.ProdConfig_Aft.Shift_StartTime + TOD_TO_UDINT(TOD#00:10:00);
		ELSIF In_From_ICxx_Pers.ProdConfig_Aft.Break1_EndTime > In_From_ICxx_Pers.ProdConfig_Aft.Shift_EndTime - TOD_TO_UDINT(TOD#00:25:00)
			THEN
				In_From_ICxx_Pers.ProdConfig_Aft.Break1_EndTime:= In_From_ICxx_Pers.ProdConfig_Aft.Shift_EndTime - TOD_TO_UDINT(TOD#00:25:00);
		(*Allow Break end time to be pushed by break start time*)
		ELSIF In_From_ICxx_Pers.ProdConfig_Aft.Break1_EndTime < In_From_ICxx_Pers.ProdConfig_Aft.Break1_StartTime + TOD_TO_UDINT(TOD#00:05:00)
			THEN
				In_From_ICxx_Pers.ProdConfig_Aft.Break1_EndTime:= In_From_ICxx_Pers.ProdConfig_Aft.Break1_StartTime + TOD_TO_UDINT(TOD#00:05:00);
		ELSIF In_From_ICxx_Pers.ProdConfig_Aft.Break1_EndTime > In_From_ICxx_Pers.ProdConfig_Aft.Break2_StartTime - TOD_TO_UDINT(TOD#00:05:00)
			THEN
				In_From_ICxx_Pers.ProdConfig_Aft.Break1_EndTime:= In_From_ICxx_Pers.ProdConfig_Aft.Break2_StartTime - TOD_TO_UDINT(TOD#00:05:00);
		END_IF;

	(*Break 2 Constraints*)
		(*Start of Break*)
		IF In_From_ICxx_Pers.ProdConfig_Aft.Break2_StartTime < In_From_ICxx_Pers.ProdConfig_Aft.Shift_StartTime + TOD_TO_UDINT(TOD#00:15:00)
			THEN
				In_From_ICxx_Pers.ProdConfig_Aft.Break2_StartTime:= In_From_ICxx_Pers.ProdConfig_Aft.Shift_StartTime + TOD_TO_UDINT(TOD#00:15:00);
		ELSIF In_From_ICxx_Pers.ProdConfig_Aft.Break2_StartTime > In_From_ICxx_Pers.ProdConfig_Aft.Shift_EndTime - TOD_TO_UDINT(TOD#00:20:00)
			THEN
				In_From_ICxx_Pers.ProdConfig_Aft.Break2_StartTime:= In_From_ICxx_Pers.ProdConfig_Aft.Shift_EndTime - TOD_TO_UDINT(TOD#00:20:00);
		ELSIF In_From_ICxx_Pers.ProdConfig_Aft.Break2_StartTime < In_From_ICxx_Pers.ProdConfig_Aft.Break1_EndTime + TOD_TO_UDINT(TOD#00:05:00)
			THEN
				In_From_ICxx_Pers.ProdConfig_Aft.Break2_StartTime:= In_From_ICxx_Pers.ProdConfig_Aft.Break1_EndTime + TOD_TO_UDINT(TOD#00:05:00);
		(*Allow Break start time to be pushed by break end time*)
		ELSIF In_From_ICxx_Pers.ProdConfig_Aft.Break2_StartTime > In_From_ICxx_Pers.ProdConfig_Aft.Break2_EndTime
			THEN
				In_From_ICxx_Pers.ProdConfig_Aft.Break2_StartTime:= In_From_ICxx_Pers.ProdConfig_Aft.Break2_EndTime - TOD_TO_UDINT(TOD#00:05:00);
		END_IF;

		(*End of Break*)
		IF In_From_ICxx_Pers.ProdConfig_Aft.Break2_EndTime < In_From_ICxx_Pers.ProdConfig_Aft.Shift_StartTime + TOD_TO_UDINT(TOD#00:20:00)
			THEN
				In_From_ICxx_Pers.ProdConfig_Aft.Break2_EndTime:= In_From_ICxx_Pers.ProdConfig_Aft.Shift_StartTime + TOD_TO_UDINT(TOD#00:20:00);
		ELSIF In_From_ICxx_Pers.ProdConfig_Aft.Break2_EndTime > In_From_ICxx_Pers.ProdConfig_Aft.Shift_EndTime - TOD_TO_UDINT(TOD#00:15:00)
			THEN
				In_From_ICxx_Pers.ProdConfig_Aft.Break2_EndTime:= In_From_ICxx_Pers.ProdConfig_Aft.Shift_EndTime - TOD_TO_UDINT(TOD#00:15:00);
		(*Allow Break end time to be pushed by break start time*)
		ELSIF In_From_ICxx_Pers.ProdConfig_Aft.Break2_EndTime < In_From_ICxx_Pers.ProdConfig_Aft.Break2_StartTime + TOD_TO_UDINT(TOD#00:05:00)
			THEN
				In_From_ICxx_Pers.ProdConfig_Aft.Break2_EndTime:= In_From_ICxx_Pers.ProdConfig_Aft.Break2_StartTime + TOD_TO_UDINT(TOD#00:05:00);
		ELSIF In_From_ICxx_Pers.ProdConfig_Aft.Break2_EndTime > In_From_ICxx_Pers.ProdConfig_Aft.Break3_StartTime - TOD_TO_UDINT(TOD#00:05:00)
			THEN
				In_From_ICxx_Pers.ProdConfig_Aft.Break2_EndTime:= In_From_ICxx_Pers.ProdConfig_Aft.Break3_StartTime - TOD_TO_UDINT(TOD#00:05:00);
		END_IF;

	(*Break 3 Constraints*)
		(*Start of Break*)
		IF In_From_ICxx_Pers.ProdConfig_Aft.Break3_StartTime < In_From_ICxx_Pers.ProdConfig_Aft.Shift_StartTime + TOD_TO_UDINT(TOD#00:20:00)
			THEN
				In_From_ICxx_Pers.ProdConfig_Aft.Break3_StartTime:= In_From_ICxx_Pers.ProdConfig_Aft.Shift_StartTime + TOD_TO_UDINT(TOD#00:20:00);
		ELSIF In_From_ICxx_Pers.ProdConfig_Aft.Break3_StartTime > In_From_ICxx_Pers.ProdConfig_Aft.Shift_EndTime - TOD_TO_UDINT(TOD#00:10:00)
			THEN
				In_From_ICxx_Pers.ProdConfig_Aft.Break3_StartTime:= In_From_ICxx_Pers.ProdConfig_Aft.Shift_EndTime - TOD_TO_UDINT(TOD#00:10:00);
		ELSIF In_From_ICxx_Pers.ProdConfig_Aft.Break3_StartTime < In_From_ICxx_Pers.ProdConfig_Aft.Break2_EndTime + TOD_TO_UDINT(TOD#00:05:00)
			THEN
				In_From_ICxx_Pers.ProdConfig_Aft.Break3_StartTime:= In_From_ICxx_Pers.ProdConfig_Aft.Break2_EndTime + TOD_TO_UDINT(TOD#00:05:00);
		(*Allow Break start time to be pushed by break end time*)
		ELSIF In_From_ICxx_Pers.ProdConfig_Aft.Break3_StartTime > In_From_ICxx_Pers.ProdConfig_Aft.Break3_EndTime
			THEN
				In_From_ICxx_Pers.ProdConfig_Aft.Break3_StartTime:= In_From_ICxx_Pers.ProdConfig_Aft.Break3_EndTime - TOD_TO_UDINT(TOD#00:05:00);
		END_IF;

		(*End of Break*)
		IF In_From_ICxx_Pers.ProdConfig_Aft.Break3_EndTime < In_From_ICxx_Pers.ProdConfig_Aft.Shift_StartTime + TOD_TO_UDINT(TOD#00:25:00)
			THEN
				In_From_ICxx_Pers.ProdConfig_Aft.Break3_EndTime:= In_From_ICxx_Pers.ProdConfig_Aft.Shift_StartTime + TOD_TO_UDINT(TOD#00:25:00);
		ELSIF In_From_ICxx_Pers.ProdConfig_Aft.Break3_EndTime > In_From_ICxx_Pers.ProdConfig_Aft.Shift_EndTime - TOD_TO_UDINT(TOD#00:05:00)
			THEN
				In_From_ICxx_Pers.ProdConfig_Aft.Break3_EndTime:= In_From_ICxx_Pers.ProdConfig_Aft.Shift_EndTime - TOD_TO_UDINT(TOD#00:05:00);
		(*Allow Break end time to be pushed by break start time*)
		ELSIF In_From_ICxx_Pers.ProdConfig_Aft.Break3_EndTime < In_From_ICxx_Pers.ProdConfig_Aft.Break3_StartTime + TOD_TO_UDINT(TOD#00:05:00)
			THEN
				In_From_ICxx_Pers.ProdConfig_Aft.Break3_EndTime:= In_From_ICxx_Pers.ProdConfig_Aft.Break3_StartTime + TOD_TO_UDINT(TOD#00:05:00);
		END_IF;


(*----------- Set Midnight Shift Constaints-------------*)
	(*Mid Shift start must fall between3pm -11pm*)
	IF UDINT_TO_TOD(In_From_ICxx_Pers.ProdConfig_Mid.Shift_StartTime) < TOD#15:00:00
		THEN
				In_From_ICxx_Pers.ProdConfig_Mid.Shift_StartTime:= TOD_TO_UDINT(TOD#15:00:00);

	ELSIF UDINT_TO_TOD(In_From_ICxx_Pers.ProdConfig_Mid.Shift_StartTime) > TOD#23:00:00
		THEN
				In_From_ICxx_Pers.ProdConfig_Mid.Shift_StartTime:= TOD_TO_UDINT(TOD#23:00:00);

	(*Midnight shift end time must fall >=1:00am (midnight shift MUST roll over midnight)*)
	ELSIF UDINT_TO_TOD(In_From_ICxx_Pers.ProdConfig_Mid.Shift_EndTime) < TOD#1:00:00
		THEN
				In_From_ICxx_Pers.ProdConfig_Mid.Shift_EndTime:= TOD_TO_UDINT(TOD#1:00:00);

	(*Set Shift maximum span as 12 hours*)
	ELSIF (86400000 - In_From_ICxx_Pers.ProdConfig_Mid.Shift_StartTime + In_From_ICxx_Pers.ProdConfig_Mid.Shift_EndTime) > 43200000 (*12 hours in UDINT form*)
		THEN
				In_From_ICxx_Pers.ProdConfig_Mid.Shift_EndTime:= (43200000 - (86400000 - In_From_ICxx_Pers.ProdConfig_Mid.Shift_StartTime));

	END_IF;

	(*Break 1 Constraints*)
		(*Start of Break*)
		IF (In_From_ICxx_Pers.ProdConfig_Mid.Break1_StartTime < In_From_ICxx_Pers.ProdConfig_Mid.Shift_StartTime + TOD_TO_UDINT(TOD#00:05:00)) AND
			In_From_ICxx_Pers.ProdConfig_Mid.Break1_StartTime > 43200000
			THEN
				In_From_ICxx_Pers.ProdConfig_Mid.Break1_StartTime:= In_From_ICxx_Pers.ProdConfig_Mid.Shift_StartTime + TOD_TO_UDINT(TOD#00:05:00);
		ELSIF (In_From_ICxx_Pers.ProdConfig_Mid.Break1_StartTime > In_From_ICxx_Pers.ProdConfig_Mid.Shift_EndTime - TOD_TO_UDINT(TOD#00:30:00)) AND
				In_From_ICxx_Pers.ProdConfig_Mid.Break1_StartTime < 43200000
			THEN
				In_From_ICxx_Pers.ProdConfig_Mid.Break1_StartTime:= In_From_ICxx_Pers.ProdConfig_Mid.Shift_EndTime - TOD_TO_UDINT(TOD#00:30:00);
		(*Allow Break start time to be pushed by break end time*)
		ELSIF (In_From_ICxx_Pers.ProdConfig_Mid.Break1_StartTime > In_From_ICxx_Pers.ProdConfig_Mid.Break1_EndTime - TOD_TO_UDINT(TOD#00:05:00)) AND
				In_From_ICxx_Pers.ProdConfig_Mid.Break1_StartTime < In_From_ICxx_Pers.ProdConfig_Mid.Shift_StartTime
			THEN
				In_From_ICxx_Pers.ProdConfig_Mid.Break1_StartTime:= In_From_ICxx_Pers.ProdConfig_Mid.Break1_EndTime - TOD_TO_UDINT(TOD#00:05:00);
			(*Midnight Rollover constraints*)
			ELSIF In_From_ICxx_Pers.ProdConfig_Mid.Break1_StartTime < 60000
				THEN
				In_From_ICxx_Pers.ProdConfig_Mid.Break1_StartTime:= 86340000;
			ELSIF In_From_ICxx_Pers.ProdConfig_Mid.Break1_StartTime > 86340000
				THEN
				In_From_ICxx_Pers.ProdConfig_Mid.Break1_StartTime:= 60000;
		END_IF;

		(*End of Break*)
		IF (In_From_ICxx_Pers.ProdConfig_Mid.Break1_EndTime < In_From_ICxx_Pers.ProdConfig_Mid.Shift_StartTime + TOD_TO_UDINT(TOD#00:10:00)) AND
			In_From_ICxx_Pers.ProdConfig_Mid.Break1_EndTime > 43200000
			THEN
				In_From_ICxx_Pers.ProdConfig_Mid.Break1_EndTime:= In_From_ICxx_Pers.ProdConfig_Mid.Shift_StartTime + TOD_TO_UDINT(TOD#00:10:00);
		ELSIF (In_From_ICxx_Pers.ProdConfig_Mid.Break1_EndTime > In_From_ICxx_Pers.ProdConfig_Mid.Shift_EndTime - TOD_TO_UDINT(TOD#00:25:00)) AND
			In_From_ICxx_Pers.ProdConfig_Mid.Break1_EndTime < 43200000
			THEN
				In_From_ICxx_Pers.ProdConfig_Mid.Break1_EndTime:= In_From_ICxx_Pers.ProdConfig_Mid.Shift_EndTime - TOD_TO_UDINT(TOD#00:25:00);
		(*Allow Break end time to be pushed by break start time*)
		ELSIF (In_From_ICxx_Pers.ProdConfig_Mid.Break1_EndTime < In_From_ICxx_Pers.ProdConfig_Mid.Break1_StartTime + TOD_TO_UDINT(TOD#00:05:00)) AND
				((In_From_ICxx_Pers.ProdConfig_Mid.Break1_EndTime < 43200000 AND  In_From_ICxx_Pers.ProdConfig_Mid.Break1_StartTime < 43200000)
				OR
				(In_From_ICxx_Pers.ProdConfig_Mid.Break1_EndTime > 43200000 AND  In_From_ICxx_Pers.ProdConfig_Mid.Break1_StartTime > 43200000))
			THEN
				In_From_ICxx_Pers.ProdConfig_Mid.Break1_EndTime:= In_From_ICxx_Pers.ProdConfig_Mid.Break1_StartTime + TOD_TO_UDINT(TOD#00:05:00);
		ELSIF (In_From_ICxx_Pers.ProdConfig_Mid.Break1_EndTime > In_From_ICxx_Pers.ProdConfig_Mid.Break2_StartTime - TOD_TO_UDINT(TOD#00:05:00)) AND
				((In_From_ICxx_Pers.ProdConfig_Mid.Break1_EndTime < 43200000 AND  In_From_ICxx_Pers.ProdConfig_Mid.Break2_StartTime < 43200000)
				OR
				(In_From_ICxx_Pers.ProdConfig_Mid.Break1_EndTime > 43200000 AND  In_From_ICxx_Pers.ProdConfig_Mid.Break2_StartTime > 43200000))
			THEN
				In_From_ICxx_Pers.ProdConfig_Mid.Break1_EndTime:= In_From_ICxx_Pers.ProdConfig_Mid.Break2_StartTime - TOD_TO_UDINT(TOD#00:05:00);
			(*Midnight Rollover constraints*)
			ELSIF In_From_ICxx_Pers.ProdConfig_Mid.Break1_EndTime < 60000
				THEN
				In_From_ICxx_Pers.ProdConfig_Mid.Break1_EndTime:= 86340000;
			ELSIF In_From_ICxx_Pers.ProdConfig_Mid.Break1_EndTime > 86340000
				THEN
				In_From_ICxx_Pers.ProdConfig_Mid.Break1_EndTime:= 60000;
		END_IF;

	(*Break 2 Constraints*)
		(*Start of Break*)
		IF (In_From_ICxx_Pers.ProdConfig_Mid.Break2_StartTime < In_From_ICxx_Pers.ProdConfig_Mid.Shift_StartTime + TOD_TO_UDINT(TOD#00:15:00)) AND
			In_From_ICxx_Pers.ProdConfig_Mid.Break2_StartTime > 43200000
			THEN
				In_From_ICxx_Pers.ProdConfig_Mid.Break2_StartTime:= In_From_ICxx_Pers.ProdConfig_Mid.Shift_StartTime + TOD_TO_UDINT(TOD#00:15:00);
		ELSIF (In_From_ICxx_Pers.ProdConfig_Mid.Break2_StartTime > In_From_ICxx_Pers.ProdConfig_Mid.Shift_EndTime - TOD_TO_UDINT(TOD#00:20:00)) AND
			In_From_ICxx_Pers.ProdConfig_Mid.Break2_StartTime < 43200000
			THEN
				In_From_ICxx_Pers.ProdConfig_Mid.Break2_StartTime:= In_From_ICxx_Pers.ProdConfig_Mid.Shift_EndTime - TOD_TO_UDINT(TOD#00:20:00);
		ELSIF (In_From_ICxx_Pers.ProdConfig_Mid.Break2_StartTime < In_From_ICxx_Pers.ProdConfig_Mid.Break1_EndTime + TOD_TO_UDINT(TOD#00:05:00)) AND
				((In_From_ICxx_Pers.ProdConfig_Mid.Break2_StartTime < 43200000 AND  In_From_ICxx_Pers.ProdConfig_Mid.Break1_EndTime < 43200000)
				OR
				(In_From_ICxx_Pers.ProdConfig_Mid.Break2_StartTime > 43200000 AND  In_From_ICxx_Pers.ProdConfig_Mid.Break1_EndTime > 43200000))
			THEN
				In_From_ICxx_Pers.ProdConfig_Mid.Break2_StartTime:= In_From_ICxx_Pers.ProdConfig_Mid.Break1_EndTime + TOD_TO_UDINT(TOD#00:05:00);
		(*Allow Break start time to be pushed by break end time*)
		ELSIF (In_From_ICxx_Pers.ProdConfig_Mid.Break2_StartTime > In_From_ICxx_Pers.ProdConfig_Mid.Break2_EndTime - TOD_TO_UDINT(TOD#00:05:00)) AND
				((In_From_ICxx_Pers.ProdConfig_Mid.Break2_StartTime < 43200000 AND  In_From_ICxx_Pers.ProdConfig_Mid.Break2_EndTime < 43200000)
				OR
				(In_From_ICxx_Pers.ProdConfig_Mid.Break2_StartTime > 43200000 AND  In_From_ICxx_Pers.ProdConfig_Mid.Break2_EndTime > 43200000))
			THEN
				In_From_ICxx_Pers.ProdConfig_Mid.Break2_StartTime:= In_From_ICxx_Pers.ProdConfig_Mid.Break2_EndTime - TOD_TO_UDINT(TOD#00:05:00);
			(*Midnight Rollover constraints*)
			ELSIF In_From_ICxx_Pers.ProdConfig_Mid.Break2_StartTime < 60000
				THEN
				In_From_ICxx_Pers.ProdConfig_Mid.Break2_StartTime:= 86340000;
			ELSIF In_From_ICxx_Pers.ProdConfig_Mid.Break2_StartTime > 86340000
				THEN
				In_From_ICxx_Pers.ProdConfig_Mid.Break2_StartTime:= 60000;
		END_IF;

		(*End of Break*)
		IF (In_From_ICxx_Pers.ProdConfig_Mid.Break2_EndTime < In_From_ICxx_Pers.ProdConfig_Mid.Shift_StartTime + TOD_TO_UDINT(TOD#00:20:00)) AND
			In_From_ICxx_Pers.ProdConfig_Mid.Break2_EndTime > 43200000
			THEN
				In_From_ICxx_Pers.ProdConfig_Mid.Break2_EndTime:= In_From_ICxx_Pers.ProdConfig_Mid.Shift_StartTime + TOD_TO_UDINT(TOD#00:20:00);
		ELSIF (In_From_ICxx_Pers.ProdConfig_Mid.Break2_EndTime > In_From_ICxx_Pers.ProdConfig_Mid.Shift_EndTime - TOD_TO_UDINT(TOD#00:15:00)) AND
			In_From_ICxx_Pers.ProdConfig_Mid.Break2_EndTime < 43200000
			THEN
				In_From_ICxx_Pers.ProdConfig_Mid.Break2_EndTime:= In_From_ICxx_Pers.ProdConfig_Mid.Shift_EndTime - TOD_TO_UDINT(TOD#00:15:00);
		(*Allow Break end time to be pushed by break start time*)
		ELSIF (In_From_ICxx_Pers.ProdConfig_Mid.Break2_EndTime < In_From_ICxx_Pers.ProdConfig_Mid.Break2_StartTime + TOD_TO_UDINT(TOD#00:05:00)) AND
				((In_From_ICxx_Pers.ProdConfig_Mid.Break2_EndTime < 43200000 AND  In_From_ICxx_Pers.ProdConfig_Mid.Break2_StartTime < 43200000)
				OR
				(In_From_ICxx_Pers.ProdConfig_Mid.Break2_EndTime > 43200000 AND  In_From_ICxx_Pers.ProdConfig_Mid.Break2_StartTime > 43200000))
			THEN
				In_From_ICxx_Pers.ProdConfig_Mid.Break2_EndTime:= In_From_ICxx_Pers.ProdConfig_Mid.Break2_StartTime + TOD_TO_UDINT(TOD#00:05:00);
		ELSIF (In_From_ICxx_Pers.ProdConfig_Mid.Break2_EndTime > In_From_ICxx_Pers.ProdConfig_Mid.Break3_StartTime - TOD_TO_UDINT(TOD#00:05:00)) AND
				((In_From_ICxx_Pers.ProdConfig_Mid.Break2_EndTime < 43200000 AND  In_From_ICxx_Pers.ProdConfig_Mid.Break3_StartTime < 43200000)
				OR
				(In_From_ICxx_Pers.ProdConfig_Mid.Break2_EndTime > 43200000 AND  In_From_ICxx_Pers.ProdConfig_Mid.Break3_StartTime > 43200000))
			THEN
				In_From_ICxx_Pers.ProdConfig_Mid.Break2_EndTime:= In_From_ICxx_Pers.ProdConfig_Mid.Break3_StartTime - TOD_TO_UDINT(TOD#00:05:00);
			(*Midnight Rollover constraints*)
			ELSIF In_From_ICxx_Pers.ProdConfig_Mid.Break2_EndTime < 60000
				THEN
				In_From_ICxx_Pers.ProdConfig_Mid.Break2_EndTime:= 86340000;
			ELSIF In_From_ICxx_Pers.ProdConfig_Mid.Break2_EndTime > 86340000
				THEN
				In_From_ICxx_Pers.ProdConfig_Mid.Break2_EndTime:= 60000;
		END_IF;

	(*Break 3 Constraints*)
		(*Start of Break*)
		IF (In_From_ICxx_Pers.ProdConfig_Mid.Break3_StartTime < In_From_ICxx_Pers.ProdConfig_Mid.Shift_StartTime + TOD_TO_UDINT(TOD#00:20:00)) AND
			In_From_ICxx_Pers.ProdConfig_Mid.Break3_StartTime > 43200000
			THEN
				In_From_ICxx_Pers.ProdConfig_Mid.Break3_StartTime:= In_From_ICxx_Pers.ProdConfig_Mid.Shift_StartTime + TOD_TO_UDINT(TOD#00:20:00);
		ELSIF (In_From_ICxx_Pers.ProdConfig_Mid.Break3_StartTime > In_From_ICxx_Pers.ProdConfig_Mid.Shift_EndTime - TOD_TO_UDINT(TOD#00:10:00)) AND
			In_From_ICxx_Pers.ProdConfig_Mid.Break3_StartTime < 43200000
			THEN
				In_From_ICxx_Pers.ProdConfig_Mid.Break3_StartTime:= In_From_ICxx_Pers.ProdConfig_Mid.Shift_EndTime - TOD_TO_UDINT(TOD#00:10:00);
		ELSIF (In_From_ICxx_Pers.ProdConfig_Mid.Break3_StartTime < In_From_ICxx_Pers.ProdConfig_Mid.Break2_EndTime + TOD_TO_UDINT(TOD#00:05:00)) AND
				((In_From_ICxx_Pers.ProdConfig_Mid.Break3_StartTime < 43200000 AND  In_From_ICxx_Pers.ProdConfig_Mid.Break2_EndTime < 43200000)
				OR
				(In_From_ICxx_Pers.ProdConfig_Mid.Break3_StartTime > 43200000 AND  In_From_ICxx_Pers.ProdConfig_Mid.Break2_EndTime > 43200000))
			THEN
				In_From_ICxx_Pers.ProdConfig_Mid.Break3_StartTime:= In_From_ICxx_Pers.ProdConfig_Mid.Break2_EndTime + TOD_TO_UDINT(TOD#00:05:00);
		(*Allow Break start time to be pushed by break end time*)
		ELSIF (In_From_ICxx_Pers.ProdConfig_Mid.Break3_StartTime > In_From_ICxx_Pers.ProdConfig_Mid.Break3_EndTime - TOD_TO_UDINT(TOD#00:05:00)) AND
				((In_From_ICxx_Pers.ProdConfig_Mid.Break3_StartTime < 43200000 AND  In_From_ICxx_Pers.ProdConfig_Mid.Break3_EndTime < 43200000)
				OR
				(In_From_ICxx_Pers.ProdConfig_Mid.Break3_StartTime > 43200000 AND  In_From_ICxx_Pers.ProdConfig_Mid.Break3_EndTime > 43200000))
			THEN
				In_From_ICxx_Pers.ProdConfig_Mid.Break3_StartTime:= In_From_ICxx_Pers.ProdConfig_Mid.Break3_EndTime - TOD_TO_UDINT(TOD#00:05:00);
			(*Midnight Rollover constraints*)
			ELSIF In_From_ICxx_Pers.ProdConfig_Mid.Break3_StartTime < 60000
				THEN
				In_From_ICxx_Pers.ProdConfig_Mid.Break3_StartTime:= 86340000;
			ELSIF In_From_ICxx_Pers.ProdConfig_Mid.Break3_StartTime > 86340000
				THEN
				In_From_ICxx_Pers.ProdConfig_Mid.Break3_StartTime:= 60000;
		END_IF;

		(*End of Break*)
		IF (In_From_ICxx_Pers.ProdConfig_Mid.Break3_EndTime < In_From_ICxx_Pers.ProdConfig_Mid.Shift_StartTime + TOD_TO_UDINT(TOD#00:25:00)) AND
			In_From_ICxx_Pers.ProdConfig_Mid.Break3_EndTime > 43200000
			THEN
				In_From_ICxx_Pers.ProdConfig_Mid.Break3_EndTime:= In_From_ICxx_Pers.ProdConfig_Mid.Shift_StartTime + TOD_TO_UDINT(TOD#00:25:00);
		ELSIF (In_From_ICxx_Pers.ProdConfig_Mid.Break3_EndTime > In_From_ICxx_Pers.ProdConfig_Mid.Shift_EndTime - TOD_TO_UDINT(TOD#00:05:00)) AND
				In_From_ICxx_Pers.ProdConfig_Mid.Break3_EndTime < 43200000
			THEN
				In_From_ICxx_Pers.ProdConfig_Mid.Break3_EndTime:= In_From_ICxx_Pers.ProdConfig_Mid.Shift_EndTime - TOD_TO_UDINT(TOD#00:05:00);
		(*Allow Break end time to be pushed by break start time*)
		ELSIF (In_From_ICxx_Pers.ProdConfig_Mid.Break3_EndTime < In_From_ICxx_Pers.ProdConfig_Mid.Break3_StartTime + TOD_TO_UDINT(TOD#00:05:00)) AND
				((In_From_ICxx_Pers.ProdConfig_Mid.Break3_EndTime < 43200000 AND  In_From_ICxx_Pers.ProdConfig_Mid.Break3_StartTime < 43200000)
				OR
				(In_From_ICxx_Pers.ProdConfig_Mid.Break3_EndTime > 43200000 AND  In_From_ICxx_Pers.ProdConfig_Mid.Break3_StartTime > 43200000))
			THEN
				In_From_ICxx_Pers.ProdConfig_Mid.Break3_EndTime:= In_From_ICxx_Pers.ProdConfig_Mid.Break3_StartTime + TOD_TO_UDINT(TOD#00:05:00);
			(*Midnight Rollover constraints*)
			ELSIF In_From_ICxx_Pers.ProdConfig_Mid.Break3_EndTime < 60000
				THEN
				In_From_ICxx_Pers.ProdConfig_Mid.Break3_EndTime:= 86340000;
			ELSIF In_From_ICxx_Pers.ProdConfig_Mid.Break3_EndTime > 86340000
				THEN
				In_From_ICxx_Pers.ProdConfig_Mid.Break3_EndTime:= 60000;
		END_IF;

(*---------- Set Shift to shift Constraints ---------------*)
	(* Ensure Day Shift's end time is not overlapping with the Aft Shift's start time*)
	IF ProdConfig_Common.Shift_Enables.2 AND
		In_From_ICxx_Pers.ProdConfig_Day.Shift_EndTime > In_From_ICxx_Pers.ProdConfig_Aft.Shift_StartTime
		THEN
				In_From_ICxx_Pers.ProdConfig_Day.Shift_EndTime:= In_From_ICxx_Pers.ProdConfig_Aft.Shift_StartTime;

	(* Ensure Aft Shift's end time is not overlapping with the Mid Shift's start time*)
	ELSIF ProdConfig_Common.Shift_Enables.3 AND
		In_From_ICxx_Pers.ProdConfig_Aft.Shift_EndTime > In_From_ICxx_Pers.ProdConfig_Mid.Shift_StartTime
		THEN
				In_From_ICxx_Pers.ProdConfig_Aft.Shift_EndTime:= In_From_ICxx_Pers.ProdConfig_Mid.Shift_StartTime;

	(* Ensure Mid Shift's end time is not overlapping with the Day Shift's start time*)
	ELSIF ProdConfig_Common.Shift_Enables.1 AND
		In_From_ICxx_Pers.ProdConfig_Mid.Shift_EndTime > In_From_ICxx_Pers.ProdConfig_Day.Shift_StartTime
		THEN
				In_From_ICxx_Pers.ProdConfig_Mid.Shift_EndTime:= In_From_ICxx_Pers.ProdConfig_Day.Shift_StartTime;

	END_IF;

(*------------- Zero Seconds Constraints ---------------*)
	(*Day Shift*)
	In_From_ICxx_Pers.ProdConfig_Day.Shift_StartTime:= FUN_GTAC_ZeroSecsInUDINT_Time(In_From_ICxx_Pers.ProdConfig_Day.Shift_StartTime);
		In_From_ICxx_Pers.ProdConfig_Day.Break1_StartTime:= FUN_GTAC_ZeroSecsInUDINT_Time(In_From_ICxx_Pers.ProdConfig_Day.Break1_StartTime);
		In_From_ICxx_Pers.ProdConfig_Day.Break1_EndTime:= FUN_GTAC_ZeroSecsInUDINT_Time(In_From_ICxx_Pers.ProdConfig_Day.Break1_EndTime);
		In_From_ICxx_Pers.ProdConfig_Day.Break2_StartTime:= FUN_GTAC_ZeroSecsInUDINT_Time(In_From_ICxx_Pers.ProdConfig_Day.Break2_StartTime);
		In_From_ICxx_Pers.ProdConfig_Day.Break2_EndTime:= FUN_GTAC_ZeroSecsInUDINT_Time(In_From_ICxx_Pers.ProdConfig_Day.Break2_EndTime);
		In_From_ICxx_Pers.ProdConfig_Day.Break3_StartTime:= FUN_GTAC_ZeroSecsInUDINT_Time(In_From_ICxx_Pers.ProdConfig_Day.Break3_StartTime);
		In_From_ICxx_Pers.ProdConfig_Day.Break3_EndTime:= FUN_GTAC_ZeroSecsInUDINT_Time(In_From_ICxx_Pers.ProdConfig_Day.Break3_EndTime);
	In_From_ICxx_Pers.ProdConfig_Day.Shift_EndTime:= FUN_GTAC_ZeroSecsInUDINT_Time(In_From_ICxx_Pers.ProdConfig_Day.Shift_EndTime);

	(*Aft Shift*)
	In_From_ICxx_Pers.ProdConfig_Aft.Shift_StartTime:= FUN_GTAC_ZeroSecsInUDINT_Time(In_From_ICxx_Pers.ProdConfig_Aft.Shift_StartTime);
		In_From_ICxx_Pers.ProdConfig_Aft.Break1_StartTime:= FUN_GTAC_ZeroSecsInUDINT_Time(In_From_ICxx_Pers.ProdConfig_Aft.Break1_StartTime);
		In_From_ICxx_Pers.ProdConfig_Aft.Break1_EndTime:= FUN_GTAC_ZeroSecsInUDINT_Time(In_From_ICxx_Pers.ProdConfig_Aft.Break1_EndTime);
		In_From_ICxx_Pers.ProdConfig_Aft.Break2_StartTime:= FUN_GTAC_ZeroSecsInUDINT_Time(In_From_ICxx_Pers.ProdConfig_Aft.Break2_StartTime);
		In_From_ICxx_Pers.ProdConfig_Aft.Break2_EndTime:= FUN_GTAC_ZeroSecsInUDINT_Time(In_From_ICxx_Pers.ProdConfig_Aft.Break2_EndTime);
		In_From_ICxx_Pers.ProdConfig_Aft.Break3_StartTime:= FUN_GTAC_ZeroSecsInUDINT_Time(In_From_ICxx_Pers.ProdConfig_Aft.Break3_StartTime);
		In_From_ICxx_Pers.ProdConfig_Aft.Break3_EndTime:= FUN_GTAC_ZeroSecsInUDINT_Time(In_From_ICxx_Pers.ProdConfig_Aft.Break3_EndTime);
	In_From_ICxx_Pers.ProdConfig_Aft.Shift_EndTime:= FUN_GTAC_ZeroSecsInUDINT_Time(In_From_ICxx_Pers.ProdConfig_Aft.Shift_EndTime);

	(*Mid Shift*)
	In_From_ICxx_Pers.ProdConfig_Mid.Shift_StartTime:= FUN_GTAC_ZeroSecsInUDINT_Time(In_From_ICxx_Pers.ProdConfig_Mid.Shift_StartTime);
		In_From_ICxx_Pers.ProdConfig_Mid.Break1_StartTime:= FUN_GTAC_ZeroSecsInUDINT_Time(In_From_ICxx_Pers.ProdConfig_Mid.Break1_StartTime);
		In_From_ICxx_Pers.ProdConfig_Mid.Break1_EndTime:= FUN_GTAC_ZeroSecsInUDINT_Time(In_From_ICxx_Pers.ProdConfig_Mid.Break1_EndTime);
		In_From_ICxx_Pers.ProdConfig_Mid.Break2_StartTime:= FUN_GTAC_ZeroSecsInUDINT_Time(In_From_ICxx_Pers.ProdConfig_Mid.Break2_StartTime);
		In_From_ICxx_Pers.ProdConfig_Mid.Break2_EndTime:= FUN_GTAC_ZeroSecsInUDINT_Time(In_From_ICxx_Pers.ProdConfig_Mid.Break2_EndTime);
		In_From_ICxx_Pers.ProdConfig_Mid.Break3_StartTime:= FUN_GTAC_ZeroSecsInUDINT_Time(In_From_ICxx_Pers.ProdConfig_Mid.Break3_StartTime);
		In_From_ICxx_Pers.ProdConfig_Mid.Break3_EndTime:= FUN_GTAC_ZeroSecsInUDINT_Time(In_From_ICxx_Pers.ProdConfig_Mid.Break3_EndTime);
	In_From_ICxx_Pers.ProdConfig_Mid.Shift_EndTime:= FUN_GTAC_ZeroSecsInUDINT_Time(In_From_ICxx_Pers.ProdConfig_Mid.Shift_EndTime);
END_ACTION

ACTION REPORTS:
(*--------------------------------------------------------------------------------------------------------------------------------------------------------*)
(* ----------------------------------------------------- Reports Action ----------------------------------------------------------------------------------*)
(*------------------------- Triggers to the UI to capture Production and Product reports and store to DB -------------------------------------------------*)
(*--------------------------------------------------------------------------------------------------------------------------------------------------------*)

(*--------- Upon first scan, blank all triggers and Acks -------------*)
IF Main.Starting_Scan_Pulse 
	THEN
	Out_To_ICxx.Production_Report_Trigger_REQS:= 0;
	In_From_ICxx.Production_Report_Trigger_ACKS:= 0;
	Out_To_ICxx.Product_Report_Trigger_REQS:= 0;
	In_From_ICxx.Product_Report_Trigger_ACKS:= 0;
END_IF;




(*-------------- Current Production Reports: Production Report Data is loaded in Fixture -> Production Action -------------*)
(*Trigger Bits 1 -16 -> Fix01 - Fix16*)
(*NOTE: Add / remove / modify as required for application, blt*)

(*Fix01*)
	IF (GTAC_Config.Option_HumanFix_Enables.1 AND Fix01.Production_Report.End_Shift_Trigger.Q)
		THEN
		(*If Fixture is enabled and generates a End of Shift pulse, set Production Report Trigger*)
		Out_To_ICxx.Production_Report_Trigger_REQS.1:= TRUE; (*Trigger bit is set False in UI script*)
	END_IF;
	
(*Fix02*)
	IF (GTAC_Config.Option_HumanFix_Enables.2 AND Fix02.Production_Report.End_Shift_Trigger.Q)
		THEN
		(*If Fixture is enabled and generates a End of Shift pulse, set Production Report Trigger*)
		Out_To_ICxx.Production_Report_Trigger_REQS.2:= TRUE; (*Trigger bit is set False in UI script*)
	END_IF;

(*Fix03*)
	IF (GTAC_Config.Option_HumanFix_Enables.3 AND Fix03.Production_Report.End_Shift_Trigger.Q)
		THEN
		(*If Fixture is enabled and generates a End of Shift pulse, set Production Report Trigger*)
		Out_To_ICxx.Production_Report_Trigger_REQS.3:= TRUE; (*Trigger bit is set False in UI script*)
	END_IF;
	
(*Fix04*)
	IF (GTAC_Config.Option_HumanFix_Enables.4 AND Fix04.Production_Report.End_Shift_Trigger.Q)
		THEN
		(*If Fixture is enabled and generates a End of Shift pulse, set Production Report Trigger*)
		Out_To_ICxx.Production_Report_Trigger_REQS.4:= TRUE; (*Trigger bit is set False in UI script*)
	END_IF;

(*Fix05*)
	IF (GTAC_Config.Option_HumanFix_Enables.5 AND Fix05.Production_Report.End_Shift_Trigger.Q)
		THEN
		(*If Fixture is enabled and generates a End of Shift pulse, set Production Report Trigger*)
		Out_To_ICxx.Production_Report_Trigger_REQS.5:= TRUE; (*Trigger bit is set False in UI script*)
	END_IF;

(*Fix06*)
	IF (GTAC_Config.Option_HumanFix_Enables.6 AND Fix06.Production_Report.End_Shift_Trigger.Q)
		THEN
		(*If Fixture is enabled and generates a End of Shift pulse, set Production Report Trigger*)
		Out_To_ICxx.Production_Report_Trigger_REQS.6:= TRUE; (*Trigger bit is set False in UI script*)
	END_IF;

(*Fix07*)
	IF (GTAC_Config.Option_HumanFix_Enables.7 AND Fix07.Production_Report.End_Shift_Trigger.Q)
		THEN
		(*If Fixture is enabled and generates a End of Shift pulse, set Production Report Trigger*)
		Out_To_ICxx.Production_Report_Trigger_REQS.7:= TRUE; (*Trigger bit is set False in UI script*)
	END_IF;

(*Fix08*)
	IF (GTAC_Config.Option_HumanFix_Enables.8 AND Fix08.Production_Report.End_Shift_Trigger.Q)
		THEN
		(*If Fixture is enabled and generates a End of Shift pulse, set Production Report Trigger*)
		Out_To_ICxx.Production_Report_Trigger_REQS.8:= TRUE; (*Trigger bit is set False in UI script*)
	END_IF;

(*Fix09*)
	IF (GTAC_Config.Option_HumanFix_Enables.9 AND Fix09.Production_Report.End_Shift_Trigger.Q)
		THEN
		(*If Fixture is enabled and generates a End of Shift pulse, set Production Report Trigger*)
		Out_To_ICxx.Production_Report_Trigger_REQS.9:= TRUE; (*Trigger bit is set False in UI script*)
	END_IF;

(*Fix10*)
	IF (GTAC_Config.Option_HumanFix_Enables.10 AND Fix10.Production_Report.End_Shift_Trigger.Q)
		THEN
		(*If Fixture is enabled and generates a End of Shift pulse, set Production Report Trigger*)
		Out_To_ICxx.Production_Report_Trigger_REQS.10:= TRUE; (*Trigger bit is set False in UI script*)
	END_IF;

(*Fix11*)
	IF (GTAC_Config.Option_HumanFix_Enables.11 AND Fix11.Production_Report.End_Shift_Trigger.Q)
		THEN
		(*If Fixture is enabled and generates a End of Shift pulse, set Production Report Trigger*)
		Out_To_ICxx.Production_Report_Trigger_REQS.11:= TRUE; (*Trigger bit is set False in UI script*)
	END_IF;

(*Fix12*)
	IF (GTAC_Config.Option_HumanFix_Enables.12 AND Fix12.Production_Report.End_Shift_Trigger.Q)
		THEN
		(*If Fixture is enabled and generates a End of Shift pulse, set Production Report Trigger*)
		Out_To_ICxx.Production_Report_Trigger_REQS.12:= TRUE; (*Trigger bit is set False in UI script*)
	END_IF;

(*Fix13*)
	IF (GTAC_Config.Option_HumanFix_Enables.13 AND Fix13.Production_Report.End_Shift_Trigger.Q)
		THEN
		(*If Fixture is enabled and generates a End of Shift pulse, set Production Report Trigger*)
		Out_To_ICxx.Production_Report_Trigger_REQS.13:= TRUE; (*Trigger bit is set False in UI script*)
	END_IF;

(*Fix14*)
	IF (GTAC_Config.Option_HumanFix_Enables.14 AND Fix14.Production_Report.End_Shift_Trigger.Q)
		THEN
		(*If Fixture is enabled and generates a End of Shift pulse, set Production Report Trigger*)
		Out_To_ICxx.Production_Report_Trigger_REQS.14:= TRUE; (*Trigger bit is set False in UI script*)
	END_IF;

(*Fix15*)
	IF (GTAC_Config.Option_HumanFix_Enables.15 AND Fix15.Production_Report.End_Shift_Trigger.Q)
		THEN
		(*If Fixture is enabled and generates a End of Shift pulse, set Production Report Trigger*)
		Out_To_ICxx.Production_Report_Trigger_REQS.15:= TRUE; (*Trigger bit is set False in UI script*)
	END_IF;
	
(*Fix16*)
	IF (GTAC_Config.Option_HumanFix_Enables.16 AND Fix16.Production_Report.End_Shift_Trigger.Q)
		THEN
		(*If Fixture is enabled and generates a End of Shift pulse, set Production Report Trigger*)
		Out_To_ICxx.Production_Report_Trigger_REQS.16:= TRUE; (*Trigger bit is set False in UI script*)
	END_IF;

	
(*------------- Customer defined Product Data Reports ---------------*) 
(*Trigger Bits 1 -16 -> Fix01 - Fix16*)
(*Trigger Bits 17 -28 -> Fix101 - Fix112*)
(*NOTE: Unfalseify / Add / Remove / Modify as required for application, blt*)

(*Fix01*)
	IF (GTAC_Config.Option_HumanFix_Enables.1 AND Fix01.Unload_Complete AND FALSE)	(*May require a different trigger depending on fixture application*)
		THEN
		(*If Fixture is enabled and generates an event indicating part is done, set Product Report Trigger*)
		Out_To_ICxx.Product_Report_Trigger_REQS.1:= TRUE; (*Trigger bit is set False in UI script*)
	END_IF;
	
(*Fix101*)
	IF ((GTAC_Config.Option_InternalFix_Count > 0) AND Fix101.Unload_Complete AND FALSE)	(*May require a different trigger depending on fixture application*)
		THEN
		(*If Fixture is enabled and generates an event indicating part is done, set Product Report Trigger*)
		Out_To_ICxx.Product_Report_Trigger_REQS.17:= TRUE; (*Trigger bit is set False in UI script*)
	END_IF;
END_ACTION

ACTION SIM:
(*--------------------------------------------------------------------------------------------------------------------------------------------------------*)
(* ----------------------------------------------------- SIM Action ----------------------------------------------------------------------------------*)
(*-------------------------  Area for SIM Specific / Work around code used during Sim based deployment -------------------------------------------------*)
(*--------------------------------------------------------------------------------------------------------------------------------------------------------*)

(*
//Sim "Start Robots" work around, used to trigger the start of all robot Master Jobs
IF GTAC_Config.In_SIM_Mode
	THEN
		(*Start all robots Operation Processing (IE Start Master Job operation or any operation called by Master) in SIM*)
		IF In_From_ICxx.StartRobots 
					 THEN
					 Main.SIM_WorkAround_StartRobots:= TRUE;
		END_IF;
		
		(*SStop all robots Operation Processing (IE Stop Master Job operation or any operation called by Master) in SIM*)
		IF In_From_ICxx.StopRobots 
					 THEN
					 Main.SIM_WorkAround_StartRobots:= FALSE;
		END_IF;
ELSE
	Main.SIM_WorkAround_StartRobots:= FALSE;
END_IF;


//Set the Boolean array true so it matches the model number. Then PRS can use this to load proper sub TOOLING based on Model selected. 
//FIX01
IF Fix01.Model_ID <> MAIN.Fix01PrevModelId THEN
    // Clear previous column
    IF (MAIN.Fix01PrevModelId >= 1) AND (MAIN.Fix01PrevModelId <= 15) THEN
        FOR MAIN.i := 1 TO 1 DO
            MAIN.SIM_WorkAround_FixNumberAndModel[MAIN.i][MAIN.Fix01PrevModelId] := FALSE;
        END_FOR
    END_IF

